  [3018] = {x=971.55, y=-22.315, z=22, rx=180, rz=141.96, shoulder=lefty, elbow=epositive, wrist=wpositive, fatherId=fReference[0]}
  [3019] = {x=972.787, y=-21.347, z=22, rx=180, rz=141.951, shoulder=lefty, elbow=epositive, wrist=wpositive, fatherId=fReference[0]}
  [3020] = {x=974.025, y=-20.378, z=22, rx=180, rz=141.942, shoulder=lefty, elbow=epositive, wrist=wpositive, fatherId=fReference[0]}
  [3021] = {x=975.263, y=-19.409, z=22, rx=180, rz=141.934, shoulder=lefty, elbow=epositive, wrist=wpositive, fatherId=fReference[0]}
  [3022] = {x=976.5, y=-18.44, z=22, rx=-180, rz=141.926, shoulder=lefty, elbow=epositive, wrist=wpositive, fatherId=fReference[0]}
  [3023] = {x=977.737, y=-17.471, z=22, rx=-180, rz=141.918, shoulder=lefty, elbow=epositive, wrist=wpositive, fatherId=fReference[0]}
  [3024] = {x=978.975, y=-16.501, z=22, rx=-180, rz=141.911, shoulder=lefty, elbow=epositive, wrist=wpositive, fatherId=fReference[0]}
  [3025] = {x=980.212, y=-15.532, z=22, rx=180, rz=141.904, shoulder=lefty, elbow=epositive, wrist=wpositive, fatherId=fReference[0]}
  [3026] = {x=981.449, y=-14.562, z=22, rx=-180, rz=141.898, shoulder=lefty, elbow=epositive, wrist=wpositive, fatherId=fReference[0]}
  [3027] = {x=982.686, y=-13.592, z=22, rx=180, rz=141.892, shoulder=lefty, elbow=epositive, wrist=wpositive, fatherId=fReference[0]}
  [3028] = {x=983.923, y=-12.621, z=22, rx=180, rz=141.887, shoulder=lefty, elbow=epositive, wrist=wpositive, fatherId=fReference[0]}
  [3029] = {x=985.16, y=-11.651, z=22, rx=-180, rz=141.882, shoulder=lefty, elbow=epositive, wrist=wpositive, fatherId=fReference[0]}
  [3030] = {x=986.397, y=-10.681, z=22, rx=180, rz=141.877, shoulder=lefty, elbow=epositive, wrist=wpositive, fatherId=fReference[0]}
  [3031] = {x=987.634, y=-9.71, z=22, rx=180, rz=141.873, shoulder=lefty, elbow=epositive, wrist=wpositive, fatherId=fReference[0]}
  [3032] = {x=988.87, y=-8.739, z=22, rx=180, rz=141.869, shoulder=lefty, elbow=epositive, wrist=wpositive, fatherId=fReference[0]}
  [3033] = {x=990.107, y=-7.769, z=22, rx=-180, rz=141.866, shoulder=lefty, elbow=epositive, wrist=wpositive, fatherId=fReference[0]}
  [3034] = {x=991.344, y=-6.798, z=22, rx=180, rz=141.863, shoulder=lefty, elbow=epositive, wrist=wpositive, fatherId=fReference[0]}
  [3035] = {x=992.58, y=-5.827, z=22, rx=-180, rz=141.86, shoulder=lefty, elbow=epositive, wrist=wpositive, fatherId=fReference[0]}
  [3036] = {x=993.817, y=-4.856, z=22, rx=180, rz=141.858, shoulder=lefty, elbow=epositive, wrist=wpositive, fatherId=fReference[0]}
  [3037] = {x=995.054, y=-3.885, z=22, rx=180, rz=141.857, shoulder=lefty, elbow=epositive, wrist=wpositive, fatherId=fReference[0]}
  [3038] = {x=996.29, y=-2.914, z=22, rx=-180, rz=141.855, shoulder=lefty, elbow=epositive, wrist=wpositive, fatherId=fReference[0]}
  [3039] = {x=997.527, y=-1.942, z=22, rx=-180, rz=141.854, shoulder=lefty, elbow=epositive, wrist=wpositive, fatherId=fReference[0]}
  [3040] = {x=998.763, y=-0.971, z=22, rx=180, rz=141.854, shoulder=lefty, elbow=epositive, wrist=wpositive, fatherId=fReference[0]}
  [3041] = {x=1000, z=22, rx=180, rz=141.854, shoulder=lefty, elbow=epositive, wrist=wpositive, fatherId=fReference[0]}
  [3042] = {x=1000, z=22, rx=180, rz=141.854, shoulder=lefty, elbow=epositive, wrist=wpositive, fatherId=fReference[0]}
  [3043] = {x=1000, z=122, rx=-180, rz=141.854, shoulder=lefty, elbow=epositive, wrist=wpositive, fatherId=fReference[0]}
  [3044] = {x=-1000, z=144, rx=180, rz=141.854, shoulder=lefty, elbow=epositive, wrist=wpositive, fatherId=fReference[0]}
  [3045] = {x=-1000, z=44, rx=180, rz=141.854, shoulder=lefty, elbow=epositive, wrist=wpositive, fatherId=fReference[0]}
  [3046] = {x=-1000, z=44, rx=180, rz=141.854, shoulder=lefty, elbow=epositive, wrist=wpositive, fatherId=fReference[0]}
  [3047] = {x=-998.763, y=0.971, z=44, rx=180, rz=141.854, shoulder=lefty, elbow=epositive, wrist=wpositive, fatherId=fReference[0]}
  [3048] = {x=-997.527, y=1.942, z=44, rx=180, rz=141.855, shoulder=lefty, elbow=epositive, wrist=wpositive, fatherId=fReference[0]}
  [3049] = {x=-996.29, y=2.914, z=44, rx=180, rz=141.857, shoulder=lefty, elbow=epositive, wrist=wpositive, fatherId=fReference[0]}
  [3050] = {x=-995.054, y=3.885, z=44, rx=180, rz=141.858, shoulder=lefty, elbow=epositive, wrist=wpositive, fatherId=fReference[0]}
  [3051] = {x=-993.817, y=4.856, z=44, rx=180, rz=141.86, shoulder=lefty, elbow=epositive, wrist=wpositive, fatherId=fReference[0]}
  [3052] = {x=-992.58, y=5.827, z=44, rx=180, rz=141.863, shoulder=lefty, elbow=epositive, wrist=wpositive, fatherId=fReference[0]}
  [3053] = {x=-991.344, y=6.798, z=44, rx=180, rz=141.866, shoulder=lefty, elbow=epositive, wrist=wpositive, fatherId=fReference[0]}
  [3054] = {x=-990.107, y=7.769, z=44, rx=180, rz=141.869, shoulder=lefty, elbow=epositive, wrist=wpositive, fatherId=fReference[0]}
  [3055] = {x=-988.87, y=8.739, z=44, rx=180, rz=141.873, shoulder=lefty, elbow=epositive, wrist=wpositive, fatherId=fReference[0]}
  [3056] = {x=-987.634, y=9.71, z=44, rx=180, rz=141.877, shoulder=lefty, elbow=epositive, wrist=wpositive, fatherId=fReference[0]}
  [3057] = {x=-986.397, y=10.681, z=44, rx=180, rz=141.882, shoulder=lefty, elbow=epositive, wrist=wpositive, fatherId=fReference[0]}
  [3058] = {x=-985.16, y=11.651, z=44, rx=180, rz=141.887, shoulder=lefty, elbow=epositive, wrist=wpositive, fatherId=fReference[0]}
  [3059] = {x=-983.923, y=12.622, z=44, rx=180, rz=141.892, shoulder=lefty, elbow=epositive, wrist=wpositive, fatherId=fReference[0]}
  [3060] = {x=-982.686, y=13.592, z=44, rx=180, rz=141.898, shoulder=lefty, elbow=epositive, wrist=wpositive, fatherId=fReference[0]}
  [3061] = {x=-981.449, y=14.562, z=44, rx=180, rz=141.904, shoulder=lefty, elbow=epositive, wrist=wpositive, fatherId=fReference[0]}
  [3062] = {x=-980.211, y=15.532, z=44, rx=180, rz=141.911, shoulder=lefty, elbow=epositive, wrist=wpositive, fatherId=fReference[0]}
  [3063] = {x=-978.974, y=16.502, z=44, rx=180, rz=141.918, shoulder=lefty, elbow=epositive, wrist=wpositive, fatherId=fReference[0]}
  [3064] = {x=-977.737, y=17.471, z=44, rx=180, rz=141.926, shoulder=lefty, elbow=epositive, wrist=wpositive, fatherId=fReference[0]}
  [3065] = {x=-976.499, y=18.441, z=44, rx=180, rz=141.934, shoulder=lefty, elbow=epositive, wrist=wpositive, fatherId=fReference[0]}
  [3066] = {x=-975.262, y=19.41, z=44, rx=180, rz=141.942, shoulder=lefty, elbow=epositive, wrist=wpositive, fatherId=fReference[0]}
  [3067] = {x=-974.024, y=20.379, z=44, rx=180, rz=141.951, shoulder=lefty, elbow=epositive, wrist=wpositive, fatherId=fReference[0]}
  [3068] = {x=-972.786, y=21.347, z=44, rx=180, rz=141.96, shoulder=lefty, elbow=epositive, wrist=wpositive, fatherId=fReference[0]}
  [3069] = {x=-971.549, y=22.316, z=44, rx=180, rz=141.97, shoulder=lefty, elbow=epositive, wrist=wpositive, fatherId=fReference[0]}
  [3070] = {x=-970.311, y=23.284, z=44, rx=180, rz=141.98, shoulder=lefty, elbow=epositive, wrist=wpositive, fatherId=fReference[0]}
  [3071] = {x=-969.072, y=24.252, z=44, rx=180, rz=141.991, shoulder=lefty, elbow=epositive, wrist=wpositive, fatherId=fReference[0]}
  [3072] = {x=-967.834, y=25.22, z=44, rx=180, rz=142.002, shoulder=lefty, elbow=epositive, wrist=wpositive, fatherId=fReference[0]}
  [3073] = {x=-966.596, y=26.187, z=44, rx=180, rz=142.013, shoulder=lefty, elbow=epositive, wrist=wpositive, fatherId=fReference[0]}
  [3074] = {x=-965.357, y=27.155, z=44, rx=180, rz=142.025, shoulder=lefty, elbow=epositive, wrist=wpositive, fatherId=fReference[0]}
  [3075] = {x=-964.119, y=28.121, z=44, rx=180, rz=142.037, shoulder=lefty, elbow=epositive, wrist=wpositive, fatherId=fReference[0]}
  [3076] = {x=-962.88, y=29.088, z=44, rx=180, rz=142.05, shoulder=lefty, elbow=epositive, wrist=wpositive, fatherId=fReference[0]}
  [3077] = {x=-961.641, y=30.054, z=44, rx=180, rz=142.063, shoulder=lefty, elbow=epositive, wrist=wpositive, fatherId=fReference[0]}
  [3078] = {x=-960.402, y=31.02, z=44, rx=180, rz=142.076, shoulder=lefty, elbow=epositive, wrist=wpositive, fatherId=fReference[0]}
  [3079] = {x=-959.163, y=31.986, z=44, rx=180, rz=142.09, shoulder=lefty, elbow=epositive, wrist=wpositive, fatherId=fReference[0]}
  [3080] = {x=-957.923, y=32.951, z=44, rx=180, rz=142.105, shoulder=lefty, elbow=epositive, wrist=wpositive, fatherId=fReference[0]}
  [3081] = {x=-956.684, y=33.916, z=44, rx=180, rz=142.12, shoulder=lefty, elbow=epositive, wrist=wpositive, fatherId=fReference[0]}
  [3082] = {x=-955.444, y=34.88, z=44, rx=180, rz=142.135, shoulder=lefty, elbow=epositive, wrist=wpositive, fatherId=fReference[0]}
  [3083] = {x=-954.204, y=35.844, z=44, rx=180, rz=142.151, shoulder=lefty, elbow=epositive, wrist=wpositive, fatherId=fReference[0]}
  [3084] = {x=-952.964, y=36.808, z=44, rx=180, rz=142.167, shoulder=lefty, elbow=epositive, wrist=wpositive, fatherId=fReference[0]}
  [3085] = {x=-951.724, y=37.771, z=44, rx=180, rz=142.183, shoulder=lefty, elbow=epositive, wrist=wpositive, fatherId=fReference[0]}
  [3086] = {x=-950.483, y=38.734, z=44, rx=180, rz=142.2, shoulder=lefty, elbow=epositive, wrist=wpositive, fatherId=fReference[0]}
  [3087] = {x=-949.243, y=39.696, z=44, rx=180, rz=142.218, shoulder=lefty, elbow=epositive, wrist=wpositive, fatherId=fReference[0]}
  [3088] = {x=-948.002, y=40.658, z=44, rx=180, rz=142.235, shoulder=lefty, elbow=epositive, wrist=wpositive, fatherId=fReference[0]}
  [3089] = {x=-946.761, y=41.619, z=44, rx=180, rz=142.254, shoulder=lefty, elbow=epositive, wrist=wpositive, fatherId=fReference[0]}
  [3090] = {x=-945.52, y=42.58, z=44, rx=180, rz=142.272, shoulder=lefty, elbow=epositive, wrist=wpositive, fatherId=fReference[0]}
  [3091] = {x=-944.278, y=43.541, z=44, rx=180, rz=142.291, shoulder=lefty, elbow=epositive, wrist=wpositive, fatherId=fReference[0]}
  [3092] = {x=-943.037, y=44.501, z=44, rx=180, rz=142.311, shoulder=lefty, elbow=epositive, wrist=wpositive, fatherId=fReference[0]}
  [3093] = {x=-941.795, y=45.46, z=44, rx=180, rz=142.331, shoulder=lefty, elbow=epositive, wrist=wpositive, fatherId=fReference[0]}
  [3094] = {x=-940.553, y=46.419, z=44, rx=180, rz=142.351, shoulder=lefty, elbow=epositive, wrist=wpositive, fatherId=fReference[0]}
  [3095] = {x=-939.31, y=47.377, z=44, rx=180, rz=142.372, shoulder=lefty, elbow=epositive, wrist=wpositive, fatherId=fReference[0]}
  [3096] = {x=-938.068, y=48.335, z=44, rx=180, rz=142.394, shoulder=lefty, elbow=epositive, wrist=wpositive, fatherId=fReference[0]}
  [3097] = {x=-936.825, y=49.292, z=44, rx=180, rz=142.415, shoulder=lefty, elbow=epositive, wrist=wpositive, fatherId=fReference[0]}
  [3098] = {x=-935.582, y=50.249, z=44, rx=180, rz=142.438, shoulder=lefty, elbow=epositive, wrist=wpositive, fatherId=fReference[0]}
  [3099] = {x=-934.339, y=51.205, z=44, rx=180, rz=142.46, shoulder=lefty, elbow=epositive, wrist=wpositive, fatherId=fReference[0]}
  [3100] = {x=-933.095, y=52.161, z=44, rx=180, rz=142.483, shoulder=lefty, elbow=epositive, wrist=wpositive, fatherId=fReference[0]}
  [3101] = {x=-931.852, y=53.116, z=44, rx=180, rz=142.507, shoulder=lefty, elbow=epositive, wrist=wpositive, fatherId=fReference[0]}
  [3102] = {x=-930.608, y=54.07, z=44, rx=-180, rz=142.531, shoulder=lefty, elbow=epositive, wrist=wpositive, fatherId=fReference[0]}
  [3103] = {x=-929.363, y=55.024, z=44, rx=180, rz=142.555, shoulder=lefty, elbow=epositive, wrist=wpositive, fatherId=fReference[0]}
  [3104] = {x=-928.119, y=55.977, z=44, rx=180, rz=142.58, shoulder=lefty, elbow=epositive, wrist=wpositive, fatherId=fReference[0]}
  [3105] = {x=-926.874, y=56.929, z=44, rx=180, rz=142.605, shoulder=lefty, elbow=epositive, wrist=wpositive, fatherId=fReference[0]}
  [3106] = {x=-925.629, y=57.881, z=44, rx=180, rz=142.631, shoulder=lefty, elbow=epositive, wrist=wpositive, fatherId=fReference[0]}
  [3107] = {x=-924.384, y=58.832, z=44, rx=180, rz=142.657, shoulder=lefty, elbow=epositive, wrist=wpositive, fatherId=fReference[0]}
  [3108] = {x=-923.138, y=59.782, z=44, rx=180, rz=142.684, shoulder=lefty, elbow=epositive, wrist=wpositive, fatherId=fReference[0]}
  [3109] = {x=-921.892, y=60.732, z=44, rx=180, rz=142.711, shoulder=lefty, elbow=epositive, wrist=wpositive, fatherId=fReference[0]}
  [3110] = {x=-920.646, y=61.681, z=44, rx=180, rz=142.738, shoulder=lefty, elbow=epositive, wrist=wpositive, fatherId=fReference[0]}
  [3111] = {x=-919.4, y=62.629, z=44, rx=180, rz=142.766, shoulder=lefty, elbow=epositive, wrist=wpositive, fatherId=fReference[0]}
  [3112] = {x=-918.153, y=63.576, z=44, rx=180, rz=142.795, shoulder=lefty, elbow=epositive, wrist=wpositive, fatherId=fReference[0]}
  [3113] = {x=-916.906, y=64.523, z=44, rx=180, rz=142.824, shoulder=lefty, elbow=epositive, wrist=wpositive, fatherId=fReference[0]}
  [3114] = {x=-915.659, y=65.469, z=44, rx=180, rz=142.853, shoulder=lefty, elbow=epositive, wrist=wpositive, fatherId=fReference[0]}
  [3115] = {x=-914.411, y=66.414, z=44, rx=180, rz=142.883, shoulder=lefty, elbow=epositive, wrist=wpositive, fatherId=fReference[0]}
  [3116] = {x=-913.163, y=67.358, z=44, rx=180, rz=142.913, shoulder=lefty, elbow=epositive, wrist=wpositive, fatherId=fReference[0]}
  [3117] = {x=-911.915, y=68.302, z=44, rx=180, rz=142.944, shoulder=lefty, elbow=epositive, wrist=wpositive, fatherId=fReference[0]}
  [3118] = {x=-910.667, y=69.245, z=44, rx=180, rz=142.975, shoulder=lefty, elbow=epositive, wrist=wpositive, fatherId=fReference[0]}
  [3119] = {x=-909.418, y=70.187, z=44, rx=180, rz=143.007, shoulder=lefty, elbow=epositive, wrist=wpositive, fatherId=fReference[0]}
  [3120] = {x=-908.169, y=71.128, z=44, rx=180, rz=143.039, shoulder=lefty, elbow=epositive, wrist=wpositive, fatherId=fReference[0]}
  [3121] = {x=-906.919, y=72.068, z=44, rx=180, rz=143.071, shoulder=lefty, elbow=epositive, wrist=wpositive, fatherId=fReference[0]}
  [3122] = {x=-905.67, y=73.007, z=44, rx=180, rz=143.104, shoulder=lefty, elbow=epositive, wrist=wpositive, fatherId=fReference[0]}
  [3123] = {x=-904.419, y=73.946, z=44, rx=180, rz=143.138, shoulder=lefty, elbow=epositive, wrist=wpositive, fatherId=fReference[0]}
  [3124] = {x=-903.169, y=74.883, z=44, rx=180, rz=143.172, shoulder=lefty, elbow=epositive, wrist=wpositive, fatherId=fReference[0]}
  [3125] = {x=-901.918, y=75.82, z=44, rx=180, rz=143.206, shoulder=lefty, elbow=epositive, wrist=wpositive, fatherId=fReference[0]}
  [3126] = {x=-900.667, y=76.756, z=44, rx=180, rz=143.241, shoulder=lefty, elbow=epositive, wrist=wpositive, fatherId=fReference[0]}
  [3127] = {x=-899.416, y=77.691, z=44, rx=180, rz=143.276, shoulder=lefty, elbow=epositive, wrist=wpositive, fatherId=fReference[0]}
  [3128] = {x=-898.164, y=78.625, z=44, rx=180, rz=143.312, shoulder=lefty, elbow=epositive, wrist=wpositive, fatherId=fReference[0]}
  [3129] = {x=-896.912, y=79.557, z=44, rx=180, rz=143.348, shoulder=lefty, elbow=epositive, wrist=wpositive, fatherId=fReference[0]}
  [3130] = {x=-895.659, y=80.489, z=44, rx=180, rz=143.385, shoulder=lefty, elbow=epositive, wrist=wpositive, fatherId=fReference[0]}
  [3131] = {x=-894.406, y=81.42, z=44, rx=180, rz=143.422, shoulder=lefty, elbow=epositive, wrist=wpositive, fatherId=fReference[0]}
  [3132] = {x=-893.153, y=82.35, z=44, rx=180, rz=143.46, shoulder=lefty, elbow=epositive, wrist=wpositive, fatherId=fReference[0]}
  [3133] = {x=-891.899, y=83.279, z=44, rx=180, rz=143.498, shoulder=lefty, elbow=epositive, wrist=wpositive, fatherId=fReference[0]}
  [3134] = {x=-890.645, y=84.207, z=44, rx=180, rz=143.536, shoulder=lefty, elbow=epositive, wrist=wpositive, fatherId=fReference[0]}
  [3135] = {x=-889.391, y=85.134, z=44, rx=180, rz=143.575, shoulder=lefty, elbow=epositive, wrist=wpositive, fatherId=fReference[0]}
  [3136] = {x=-888.136, y=86.06, z=44, rx=180, rz=143.615, shoulder=lefty, elbow=epositive, wrist=wpositive, fatherId=fReference[0]}
  [3137] = {x=-886.881, y=86.985, z=44, rx=180, rz=143.655, shoulder=lefty, elbow=epositive, wrist=wpositive, fatherId=fReference[0]}
  [3138] = {x=-885.626, y=87.909, z=44, rx=180, rz=143.696, shoulder=lefty, elbow=epositive, wrist=wpositive, fatherId=fReference[0]}
  [3139] = {x=-884.37, y=88.832, z=44, rx=180, rz=143.737, shoulder=lefty, elbow=epositive, wrist=wpositive, fatherId=fReference[0]}
  [3140] = {x=-883.113, y=89.753, z=44, rx=180, rz=143.778, shoulder=lefty, elbow=epositive, wrist=wpositive, fatherId=fReference[0]}
  [3141] = {x=-881.857, y=90.674, z=44, rx=180, rz=143.82, shoulder=lefty, elbow=epositive, wrist=wpositive, fatherId=fReference[0]}
  [3142] = {x=-880.6, y=91.593, z=44, rx=180, rz=143.862, shoulder=lefty, elbow=epositive, wrist=wpositive, fatherId=fReference[0]}
  [3143] = {x=-879.342, y=92.511, z=44, rx=180, rz=143.905, shoulder=lefty, elbow=epositive, wrist=wpositive, fatherId=fReference[0]}
  [3144] = {x=-878.084, y=93.428, z=44, rx=180, rz=143.949, shoulder=lefty, elbow=epositive, wrist=wpositive, fatherId=fReference[0]}
  [3145] = {x=-876.826, y=94.344, z=44, rx=180, rz=143.993, shoulder=lefty, elbow=epositive, wrist=wpositive, fatherId=fReference[0]}
  [3146] = {x=-875.567, y=95.259, z=44, rx=180, rz=144.037, shoulder=lefty, elbow=epositive, wrist=wpositive, fatherId=fReference[0]}
  [3147] = {x=-874.308, y=96.173, z=44, rx=180, rz=144.082, shoulder=lefty, elbow=epositive, wrist=wpositive, fatherId=fReference[0]}
  [3148] = {x=-873.049, y=97.085, z=44, rx=180, rz=144.127, shoulder=lefty, elbow=epositive, wrist=wpositive, fatherId=fReference[0]}
  [3149] = {x=-871.789, y=97.996, z=44, rx=180, rz=144.173, shoulder=lefty, elbow=epositive, wrist=wpositive, fatherId=fReference[0]}
  [3150] = {x=-870.528, y=98.906, z=44, rx=180, rz=144.22, shoulder=lefty, elbow=epositive, wrist=wpositive, fatherId=fReference[0]}
  [3151] = {x=-869.267, y=99.815, z=44, rx=-180, rz=144.266, shoulder=lefty, elbow=epositive, wrist=wpositive, fatherId=fReference[0]}
  [3152] = {x=-868.006, y=100.722, z=44, rx=180, rz=144.314, shoulder=lefty, elbow=epositive, wrist=wpositive, fatherId=fReference[0]}
  [3153] = {x=-866.745, y=101.628, z=44, rx=180, rz=144.362, shoulder=lefty, elbow=epositive, wrist=wpositive, fatherId=fReference[0]}
  [3154] = {x=-865.482, y=102.533, z=44, rx=180, rz=144.41, shoulder=lefty, elbow=epositive, wrist=wpositive, fatherId=fReference[0]}
  [3155] = {x=-864.22, y=103.437, z=44, rx=180, rz=144.459, shoulder=lefty, elbow=epositive, wrist=wpositive, fatherId=fReference[0]}
  [3156] = {x=-862.957, y=104.339, z=44, rx=180, rz=144.508, shoulder=lefty, elbow=epositive, wrist=wpositive, fatherId=fReference[0]}
  [3157] = {x=-861.693, y=105.24, z=44, rx=180, rz=144.558, shoulder=lefty, elbow=epositive, wrist=wpositive, fatherId=fReference[0]}
  [3158] = {x=-860.429, y=106.139, z=44, rx=180, rz=144.609, shoulder=lefty, elbow=epositive, wrist=wpositive, fatherId=fReference[0]}
  [3159] = {x=-859.165, y=107.038, z=44, rx=180, rz=144.659, shoulder=lefty, elbow=epositive, wrist=wpositive, fatherId=fReference[0]}
  [3160] = {x=-857.9, y=107.935, z=44, rx=180, rz=144.711, shoulder=lefty, elbow=epositive, wrist=wpositive, fatherId=fReference[0]}
  [3161] = {x=-856.635, y=108.83, z=44, rx=180, rz=144.763, shoulder=lefty, elbow=epositive, wrist=wpositive, fatherId=fReference[0]}
  [3162] = {x=-855.369, y=109.724, z=44, rx=180, rz=144.815, shoulder=lefty, elbow=epositive, wrist=wpositive, fatherId=fReference[0]}
  [3163] = {x=-854.103, y=110.617, z=44, rx=180, rz=144.868, shoulder=lefty, elbow=epositive, wrist=wpositive, fatherId=fReference[0]}
  [3164] = {x=-852.836, y=111.508, z=44, rx=180, rz=144.922, shoulder=lefty, elbow=epositive, wrist=wpositive, fatherId=fReference[0]}
  [3165] = {x=-851.569, y=112.398, z=44, rx=180, rz=144.976, shoulder=lefty, elbow=epositive, wrist=wpositive, fatherId=fReference[0]}
  [3166] = {x=-850.301, y=113.287, z=44, rx=180, rz=145.03, shoulder=lefty, elbow=epositive, wrist=wpositive, fatherId=fReference[0]}
  [3167] = {x=-849.033, y=114.174, z=44, rx=180, rz=145.085, shoulder=lefty, elbow=epositive, wrist=wpositive, fatherId=fReference[0]}
  [3168] = {x=-847.764, y=115.059, z=44, rx=180, rz=145.141, shoulder=lefty, elbow=epositive, wrist=wpositive, fatherId=fReference[0]}
  [3169] = {x=-846.495, y=115.943, z=44, rx=180, rz=145.197, shoulder=lefty, elbow=epositive, wrist=wpositive, fatherId=fReference[0]}
  [3170] = {x=-845.225, y=116.826, z=44, rx=180, rz=145.253, shoulder=lefty, elbow=epositive, wrist=wpositive, fatherId=fReference[0]}
  [3171] = {x=-843.955, y=117.707, z=44, rx=180, rz=145.311, shoulder=lefty, elbow=epositive, wrist=wpositive, fatherId=fReference[0]}
  [3172] = {x=-842.685, y=118.586, z=44, rx=180, rz=145.368, shoulder=lefty, elbow=epositive, wrist=wpositive, fatherId=fReference[0]}
  [3173] = {x=-841.413, y=119.464, z=44, rx=180, rz=145.426, shoulder=lefty, elbow=epositive, wrist=wpositive, fatherId=fReference[0]}
  [3174] = {x=-840.142, y=120.341, z=44, rx=180, rz=145.485, shoulder=lefty, elbow=epositive, wrist=wpositive, fatherId=fReference[0]}
  [3175] = {x=-838.869, y=121.216, z=44, rx=180, rz=145.544, shoulder=lefty, elbow=epositive, wrist=wpositive, fatherId=fReference[0]}
  [3176] = {x=-837.597, y=122.089, z=44, rx=180, rz=145.604, shoulder=lefty, elbow=epositive, wrist=wpositive, fatherId=fReference[0]}
  [3177] = {x=-836.323, y=122.961, z=44, rx=180, rz=145.665, shoulder=lefty, elbow=epositive, wrist=wpositive, fatherId=fReference[0]}
  [3178] = {x=-835.049, y=123.831, z=44, rx=180, rz=145.725, shoulder=lefty, elbow=epositive, wrist=wpositive, fatherId=fReference[0]}
  [3179] = {x=-833.775, y=124.699, z=44, rx=180, rz=145.787, shoulder=lefty, elbow=epositive, wrist=wpositive, fatherId=fReference[0]}
  [3180] = {x=-832.5, y=125.566, z=44, rx=180, rz=145.849, shoulder=lefty, elbow=epositive, wrist=wpositive, fatherId=fReference[0]}
  [3181] = {x=-831.225, y=126.431, z=44, rx=180, rz=145.911, shoulder=lefty, elbow=epositive, wrist=wpositive, fatherId=fReference[0]}
  [3182] = {x=-829.949, y=127.295, z=44, rx=180, rz=145.974, shoulder=lefty, elbow=epositive, wrist=wpositive, fatherId=fReference[0]}
  [3183] = {x=-828.672, y=128.157, z=44, rx=180, rz=146.038, shoulder=lefty, elbow=epositive, wrist=wpositive, fatherId=fReference[0]}
  [3184] = {x=-827.395, y=129.017, z=44, rx=180, rz=146.102, shoulder=lefty, elbow=epositive, wrist=wpositive, fatherId=fReference[0]}
  [3185] = {x=-826.117, y=129.876, z=44, rx=180, rz=146.167, shoulder=lefty, elbow=epositive, wrist=wpositive, fatherId=fReference[0]}
  [3186] = {x=-824.839, y=130.732, z=44, rx=180, rz=146.232, shoulder=lefty, elbow=epositive, wrist=wpositive, fatherId=fReference[0]}
  [3187] = {x=-823.56, y=131.587, z=44, rx=180, rz=146.298, shoulder=lefty, elbow=epositive, wrist=wpositive, fatherId=fReference[0]}
  [3188] = {x=-822.281, y=132.441, z=44, rx=180, rz=146.364, shoulder=lefty, elbow=epositive, wrist=wpositive, fatherId=fReference[0]}
  [3189] = {x=-821.001, y=133.292, z=44, rx=180, rz=146.431, shoulder=lefty, elbow=epositive, wrist=wpositive, fatherId=fReference[0]}
  [3190] = {x=-819.721, y=134.142, z=44, rx=180, rz=146.499, shoulder=lefty, elbow=epositive, wrist=wpositive, fatherId=fReference[0]}
  [3191] = {x=-818.44, y=134.99, z=44, rx=180, rz=146.567, shoulder=lefty, elbow=epositive, wrist=wpositive, fatherId=fReference[0]}
  [3192] = {x=-817.158, y=135.836, z=44, rx=180, rz=146.636, shoulder=lefty, elbow=epositive, wrist=wpositive, fatherId=fReference[0]}
  [3193] = {x=-815.876, y=136.68, z=44, rx=180, rz=146.705, shoulder=lefty, elbow=epositive, wrist=wpositive, fatherId=fReference[0]}
  [3194] = {x=-814.593, y=137.523, z=44, rx=180, rz=146.775, shoulder=lefty, elbow=epositive, wrist=wpositive, fatherId=fReference[0]}
  [3195] = {x=-813.309, y=138.364, z=44, rx=180, rz=146.845, shoulder=lefty, elbow=epositive, wrist=wpositive, fatherId=fReference[0]}
  [3196] = {x=-812.025, y=139.202, z=44, rx=180, rz=146.916, shoulder=lefty, elbow=epositive, wrist=wpositive, fatherId=fReference[0]}
  [3197] = {x=-810.74, y=140.039, z=44, rx=180, rz=146.987, shoulder=lefty, elbow=epositive, wrist=wpositive, fatherId=fReference[0]}
  [3198] = {x=-809.455, y=140.875, z=44, rx=180, rz=147.059, shoulder=lefty, elbow=epositive, wrist=wpositive, fatherId=fReference[0]}
  [3199] = {x=-808.169, y=141.708, z=44, rx=180, rz=147.132, shoulder=lefty, elbow=epositive, wrist=wpositive, fatherId=fReference[0]}
  [3200] = {x=-806.883, y=142.539, z=44, rx=180, rz=147.205, shoulder=lefty, elbow=epositive, wrist=wpositive, fatherId=fReference[0]}
  [3201] = {x=-805.596, y=143.368, z=44, rx=180, rz=147.279, shoulder=lefty, elbow=epositive, wrist=wpositive, fatherId=fReference[0]}
  [3202] = {x=-804.308, y=144.196, z=44, rx=180, rz=147.353, shoulder=lefty, elbow=epositive, wrist=wpositive, fatherId=fReference[0]}
  [3203] = {x=-803.019, y=145.021, z=44, rx=180, rz=147.428, shoulder=lefty, elbow=epositive, wrist=wpositive, fatherId=fReference[0]}
  [3204] = {x=-801.73, y=145.845, z=44, rx=180, rz=147.504, shoulder=lefty, elbow=epositive, wrist=wpositive, fatherId=fReference[0]}
  [3205] = {x=-800.44, y=146.666, z=44, rx=180, rz=147.58, shoulder=lefty, elbow=epositive, wrist=wpositive, fatherId=fReference[0]}
  [3206] = {x=-799.15, y=147.486, z=44, rx=180, rz=147.657, shoulder=lefty, elbow=epositive, wrist=wpositive, fatherId=fReference[0]}
  [3207] = {x=-797.859, y=148.303, z=44, rx=180, rz=147.734, shoulder=lefty, elbow=epositive, wrist=wpositive, fatherId=fReference[0]}
  [3208] = {x=-796.567, y=149.119, z=44, rx=180, rz=147.812, shoulder=lefty, elbow=epositive, wrist=wpositive, fatherId=fReference[0]}
  [3209] = {x=-795.275, y=149.932, z=44, rx=180, rz=147.891, shoulder=lefty, elbow=epositive, wrist=wpositive, fatherId=fReference[0]}
  [3210] = {x=-793.982, y=150.744, z=44, rx=180, rz=147.97, shoulder=lefty, elbow=epositive, wrist=wpositive, fatherId=fReference[0]}
  [3211] = {x=-792.688, y=151.553, z=44, rx=180, rz=148.05, shoulder=lefty, elbow=epositive, wrist=wpositive, fatherId=fReference[0]}
  [3212] = {x=-791.394, y=152.36, z=44, rx=180, rz=148.13, shoulder=lefty, elbow=epositive, wrist=wpositive, fatherId=fReference[0]}
  [3213] = {x=-790.099, y=153.165, z=44, rx=180, rz=148.211, shoulder=lefty, elbow=epositive, wrist=wpositive, fatherId=fReference[0]}
  [3214] = {x=-788.803, y=153.968, z=44, rx=180, rz=148.293, shoulder=lefty, elbow=epositive, wrist=wpositive, fatherId=fReference[0]}
  [3215] = {x=-787.507, y=154.769, z=44, rx=180, rz=148.375, shoulder=lefty, elbow=epositive, wrist=wpositive, fatherId=fReference[0]}
  [3216] = {x=-786.21, y=155.568, z=44, rx=180, rz=148.458, shoulder=lefty, elbow=epositive, wrist=wpositive, fatherId=fReference[0]}
  [3217] = {x=-784.912, y=156.365, z=44, rx=180, rz=148.541, shoulder=lefty, elbow=epositive, wrist=wpositive, fatherId=fReference[0]}
  [3218] = {x=-783.613, y=157.159, z=44, rx=180, rz=148.625, shoulder=lefty, elbow=epositive, wrist=wpositive, fatherId=fReference[0]}
  [3219] = {x=-782.314, y=157.951, z=44, rx=180, rz=148.71, shoulder=lefty, elbow=epositive, wrist=wpositive, fatherId=fReference[0]}
  [3220] = {x=-781.014, y=158.741, z=44, rx=180, rz=148.795, shoulder=lefty, elbow=epositive, wrist=wpositive, fatherId=fReference[0]}
  [3221] = {x=-779.714, y=159.529, z=44, rx=180, rz=148.881, shoulder=lefty, elbow=epositive, wrist=wpositive, fatherId=fReference[0]}
  [3222] = {x=-778.413, y=160.315, z=44, rx=180, rz=148.968, shoulder=lefty, elbow=epositive, wrist=wpositive, fatherId=fReference[0]}
  [3223] = {x=-777.111, y=161.098, z=44, rx=180, rz=149.055, shoulder=lefty, elbow=epositive, wrist=wpositive, fatherId=fReference[0]}
  [3224] = {x=-775.808, y=161.879, z=44, rx=180, rz=149.143, shoulder=lefty, elbow=epositive, wrist=wpositive, fatherId=fReference[0]}
  [3225] = {x=-774.505, y=162.658, z=44, rx=180, rz=149.231, shoulder=lefty, elbow=epositive, wrist=wpositive, fatherId=fReference[0]}
  [3226] = {x=-773.2, y=163.434, z=44, rx=180, rz=149.32, shoulder=lefty, elbow=epositive, wrist=wpositive, fatherId=fReference[0]}
  [3227] = {x=-771.896, y=164.208, z=44, rx=180, rz=149.41, shoulder=lefty, elbow=epositive, wrist=wpositive, fatherId=fReference[0]}
  [3228] = {x=-770.59, y=164.98, z=44, rx=180, rz=149.5, shoulder=lefty, elbow=epositive, wrist=wpositive, fatherId=fReference[0]}
  [3229] = {x=-769.284, y=165.75, z=44, rx=-180, rz=149.591, shoulder=lefty, elbow=epositive, wrist=wpositive, fatherId=fReference[0]}
  [3230] = {x=-767.977, y=166.517, z=44, rx=180, rz=149.683, shoulder=lefty, elbow=epositive, wrist=wpositive, fatherId=fReference[0]}
  [3231] = {x=-766.669, y=167.281, z=44, rx=180, rz=149.775, shoulder=lefty, elbow=epositive, wrist=wpositive, fatherId=fReference[0]}
  [3232] = {x=-765.36, y=168.044, z=44, rx=180, rz=149.868, shoulder=lefty, elbow=epositive, wrist=wpositive, fatherId=fReference[0]}
  [3233] = {x=-764.051, y=168.804, z=44, rx=180, rz=149.962, shoulder=lefty, elbow=epositive, wrist=wpositive, fatherId=fReference[0]}
  [3234] = {x=-762.741, y=169.561, z=44, rx=180, rz=150.056, shoulder=lefty, elbow=epositive, wrist=wpositive, fatherId=fReference[0]}
  [3235] = {x=-761.431, y=170.316, z=44, rx=180, rz=150.151, shoulder=lefty, elbow=epositive, wrist=wpositive, fatherId=fReference[0]}
  [3236] = {x=-760.119, y=171.069, z=44, rx=180, rz=150.247, shoulder=lefty, elbow=epositive, wrist=wpositive, fatherId=fReference[0]}
  [3237] = {x=-758.807, y=171.819, z=44, rx=-180, rz=150.343, shoulder=lefty, elbow=epositive, wrist=wpositive, fatherId=fReference[0]}
  [3238] = {x=-757.494, y=172.566, z=44, rx=180, rz=150.44, shoulder=lefty, elbow=epositive, wrist=wpositive, fatherId=fReference[0]}
  [3239] = {x=-756.181, y=173.311, z=44, rx=180, rz=150.537, shoulder=lefty, elbow=epositive, wrist=wpositive, fatherId=fReference[0]}
  [3240] = {x=-754.866, y=174.054, z=44, rx=180, rz=150.636, shoulder=lefty, elbow=epositive, wrist=wpositive, fatherId=fReference[0]}
  [3241] = {x=-753.551, y=174.794, z=44, rx=180, rz=150.734, shoulder=lefty, elbow=epositive, wrist=wpositive, fatherId=fReference[0]}
  [3242] = {x=-752.235, y=175.531, z=44, rx=-180, rz=150.834, shoulder=lefty, elbow=epositive, wrist=wpositive, fatherId=fReference[0]}
  [3243] = {x=-750.919, y=176.266, z=44, rx=-180, rz=150.934, shoulder=lefty, elbow=epositive, wrist=wpositive, fatherId=fReference[0]}
  [3244] = {x=-749.601, y=176.998, z=44, rx=180, rz=151.035, shoulder=lefty, elbow=epositive, wrist=wpositive, fatherId=fReference[0]}
  [3245] = {x=-748.283, y=177.727, z=44, rx=180, rz=151.137, shoulder=lefty, elbow=epositive, wrist=wpositive, fatherId=fReference[0]}
  [3246] = {x=-746.965, y=178.454, z=44, rx=180, rz=151.239, shoulder=lefty, elbow=epositive, wrist=wpositive, fatherId=fReference[0]}
  [3247] = {x=-745.645, y=179.179, z=44, rx=180, rz=151.342, shoulder=lefty, elbow=epositive, wrist=wpositive, fatherId=fReference[0]}
  [3248] = {x=-744.325, y=179.9, z=44, rx=-180, rz=151.445, shoulder=lefty, elbow=epositive, wrist=wpositive, fatherId=fReference[0]}
  [3249] = {x=-743.004, y=180.619, z=44, rx=180, rz=151.549, shoulder=lefty, elbow=epositive, wrist=wpositive, fatherId=fReference[0]}
  [3250] = {x=-741.682, y=181.335, z=44, rx=180, rz=151.654, shoulder=lefty, elbow=epositive, wrist=wpositive, fatherId=fReference[0]}
  [3251] = {x=-740.359, y=182.049, z=44, rx=180, rz=151.76, shoulder=lefty, elbow=epositive, wrist=wpositive, fatherId=fReference[0]}
  [3252] = {x=-739.036, y=182.76, z=44, rx=180, rz=151.866, shoulder=lefty, elbow=epositive, wrist=wpositive, fatherId=fReference[0]}
  [3253] = {x=-737.712, y=183.468, z=44, rx=180, rz=151.973, shoulder=lefty, elbow=epositive, wrist=wpositive, fatherId=fReference[0]}
  [3254] = {x=-736.387, y=184.173, z=44, rx=180, rz=152.081, shoulder=lefty, elbow=epositive, wrist=wpositive, fatherId=fReference[0]}
  [3255] = {x=-735.061, y=184.875, z=44, rx=180, rz=152.189, shoulder=lefty, elbow=epositive, wrist=wpositive, fatherId=fReference[0]}
  [3256] = {x=-733.735, y=185.575, z=44, rx=180, rz=152.298, shoulder=lefty, elbow=epositive, wrist=wpositive, fatherId=fReference[0]}
  [3257] = {x=-732.408, y=186.272, z=44, rx=180, rz=152.408, shoulder=lefty, elbow=epositive, wrist=wpositive, fatherId=fReference[0]}
  [3258] = {x=-731.08, y=186.966, z=44, rx=-180, rz=152.518, shoulder=lefty, elbow=epositive, wrist=wpositive, fatherId=fReference[0]}
  [3259] = {x=-729.751, y=187.657, z=44, rx=180, rz=152.63, shoulder=lefty, elbow=epositive, wrist=wpositive, fatherId=fReference[0]}
  [3260] = {x=-728.422, y=188.345, z=44, rx=180, rz=152.741, shoulder=lefty, elbow=epositive, wrist=wpositive, fatherId=fReference[0]}
  [3261] = {x=-727.092, y=189.03, z=44, rx=180, rz=152.854, shoulder=lefty, elbow=epositive, wrist=wpositive, fatherId=fReference[0]}
  [3262] = {x=-725.761, y=189.713, z=44, rx=180, rz=152.967, shoulder=lefty, elbow=epositive, wrist=wpositive, fatherId=fReference[0]}
  [3263] = {x=-724.429, y=190.392, z=44, rx=180, rz=153.081, shoulder=lefty, elbow=epositive, wrist=wpositive, fatherId=fReference[0]}
  [3264] = {x=-723.097, y=191.069, z=44, rx=180, rz=153.196, shoulder=lefty, elbow=epositive, wrist=wpositive, fatherId=fReference[0]}
  [3265] = {x=-721.764, y=191.742, z=44, rx=180, rz=153.311, shoulder=lefty, elbow=epositive, wrist=wpositive, fatherId=fReference[0]}
  [3266] = {x=-720.43, y=192.413, z=44, rx=180, rz=153.427, shoulder=lefty, elbow=epositive, wrist=wpositive, fatherId=fReference[0]}
  [3267] = {x=-719.095, y=193.08, z=44, rx=180, rz=153.544, shoulder=lefty, elbow=epositive, wrist=wpositive, fatherId=fReference[0]}
  [3268] = {x=-717.76, y=193.745, z=44, rx=180, rz=153.661, shoulder=lefty, elbow=epositive, wrist=wpositive, fatherId=fReference[0]}
  [3269] = {x=-716.424, y=194.406, z=44, rx=180, rz=153.779, shoulder=lefty, elbow=epositive, wrist=wpositive, fatherId=fReference[0]}
  [3270] = {x=-715.087, y=195.065, z=44, rx=180, rz=153.898, shoulder=lefty, elbow=epositive, wrist=wpositive, fatherId=fReference[0]}
  [3271] = {x=-713.749, y=195.72, z=44, rx=180, rz=154.017, shoulder=lefty, elbow=epositive, wrist=wpositive, fatherId=fReference[0]}
  [3272] = {x=-712.411, y=196.372, z=44, rx=180, rz=154.138, shoulder=lefty, elbow=epositive, wrist=wpositive, fatherId=fReference[0]}
  [3273] = {x=-711.072, y=197.022, z=44, rx=180, rz=154.259, shoulder=lefty, elbow=epositive, wrist=wpositive, fatherId=fReference[0]}
  [3274] = {x=-709.732, y=197.668, z=44, rx=180, rz=154.38, shoulder=lefty, elbow=epositive, wrist=wpositive, fatherId=fReference[0]}
  [3275] = {x=-708.391, y=198.311, z=44, rx=180, rz=154.503, shoulder=lefty, elbow=epositive, wrist=wpositive, fatherId=fReference[0]}
  [3276] = {x=-707.05, y=198.95, z=44, rx=-180, rz=154.626, shoulder=lefty, elbow=epositive, wrist=wpositive, fatherId=fReference[0]}
  [3277] = {x=-705.708, y=199.587, z=44, rx=180, rz=154.75, shoulder=lefty, elbow=epositive, wrist=wpositive, fatherId=fReference[0]}
  [3278] = {x=-704.365, y=200.22, z=44, rx=180, rz=154.874, shoulder=lefty, elbow=epositive, wrist=wpositive, fatherId=fReference[0]}
  [3279] = {x=-703.021, y=200.85, z=44, rx=180, rz=154.999, shoulder=lefty, elbow=epositive, wrist=wpositive, fatherId=fReference[0]}
  [3280] = {x=-701.677, y=201.477, z=44, rx=180, rz=155.125, shoulder=lefty, elbow=epositive, wrist=wpositive, fatherId=fReference[0]}
  [3281] = {x=-700.332, y=202.101, z=44, rx=180, rz=155.252, shoulder=lefty, elbow=epositive, wrist=wpositive, fatherId=fReference[0]}
  [3282] = {x=-698.986, y=202.721, z=44, rx=180, rz=155.379, shoulder=lefty, elbow=epositive, wrist=wpositive, fatherId=fReference[0]}
  [3283] = {x=-697.639, y=203.338, z=44, rx=180, rz=155.508, shoulder=lefty, elbow=epositive, wrist=wpositive, fatherId=fReference[0]}
  [3284] = {x=-696.292, y=203.952, z=44, rx=-180, rz=155.636, shoulder=lefty, elbow=epositive, wrist=wpositive, fatherId=fReference[0]}
  [3285] = {x=-694.944, y=204.563, z=44, rx=180, rz=155.766, shoulder=lefty, elbow=epositive, wrist=wpositive, fatherId=fReference[0]}
  [3286] = {x=-693.595, y=205.17, z=44, rx=180, rz=155.896, shoulder=lefty, elbow=epositive, wrist=wpositive, fatherId=fReference[0]}
  [3287] = {x=-692.246, y=205.774, z=44, rx=180, rz=156.027, shoulder=lefty, elbow=epositive, wrist=wpositive, fatherId=fReference[0]}
  [3288] = {x=-690.895, y=206.374, z=44, rx=180, rz=156.159, shoulder=lefty, elbow=epositive, wrist=wpositive, fatherId=fReference[0]}
  [3289] = {x=-689.544, y=206.971, z=44, rx=180, rz=156.291, shoulder=lefty, elbow=epositive, wrist=wpositive, fatherId=fReference[0]}
  [3290] = {x=-688.193, y=207.565, z=44, rx=-180, rz=156.425, shoulder=lefty, elbow=epositive, wrist=wpositive, fatherId=fReference[0]}
  [3291] = {x=-686.84, y=208.155, z=44, rx=180, rz=156.559, shoulder=lefty, elbow=epositive, wrist=wpositive, fatherId=fReference[0]}
  [3292] = {x=-685.487, y=208.741, z=44, rx=180, rz=156.693, shoulder=lefty, elbow=epositive, wrist=wpositive, fatherId=fReference[0]}
  [3293] = {x=-684.133, y=209.325, z=44, rx=180, rz=156.828, shoulder=lefty, elbow=epositive, wrist=wpositive, fatherId=fReference[0]}
  [3294] = {x=-682.778, y=209.905, z=44, rx=180, rz=156.965, shoulder=lefty, elbow=epositive, wrist=wpositive, fatherId=fReference[0]}
  [3295] = {x=-681.423, y=210.481, z=44, rx=180, rz=157.101, shoulder=lefty, elbow=epositive, wrist=wpositive, fatherId=fReference[0]}
  [3296] = {x=-680.067, y=211.054, z=44, rx=-180, rz=157.239, shoulder=lefty, elbow=epositive, wrist=wpositive, fatherId=fReference[0]}
  [3297] = {x=-678.71, y=211.623, z=44, rx=180, rz=157.377, shoulder=lefty, elbow=epositive, wrist=wpositive, fatherId=fReference[0]}
  [3298] = {x=-677.353, y=212.189, z=44, rx=-180, rz=157.516, shoulder=lefty, elbow=epositive, wrist=wpositive, fatherId=fReference[0]}
  [3299] = {x=-675.994, y=212.751, z=44, rx=-180, rz=157.656, shoulder=lefty, elbow=epositive, wrist=wpositive, fatherId=fReference[0]}
  [3300] = {x=-674.635, y=213.309, z=44, rx=180, rz=157.796, shoulder=lefty, elbow=epositive, wrist=wpositive, fatherId=fReference[0]}
  [3301] = {x=-673.276, y=213.864, z=44, rx=180, rz=157.937, shoulder=lefty, elbow=epositive, wrist=wpositive, fatherId=fReference[0]}
  [3302] = {x=-671.915, y=214.416, z=44, rx=180, rz=158.079, shoulder=lefty, elbow=epositive, wrist=wpositive, fatherId=fReference[0]}
  [3303] = {x=-670.554, y=214.963, z=44, rx=180, rz=158.222, shoulder=lefty, elbow=epositive, wrist=wpositive, fatherId=fReference[0]}
  [3304] = {x=-669.193, y=215.508, z=44, rx=180, rz=158.365, shoulder=lefty, elbow=epositive, wrist=wpositive, fatherId=fReference[0]}
  [3305] = {x=-667.83, y=216.048, z=44, rx=-180, rz=158.509, shoulder=lefty, elbow=epositive, wrist=wpositive, fatherId=fReference[0]}
  [3306] = {x=-666.467, y=216.585, z=44, rx=180, rz=158.654, shoulder=lefty, elbow=epositive, wrist=wpositive, fatherId=fReference[0]}
  [3307] = {x=-665.103, y=217.118, z=44, rx=180, rz=158.799, shoulder=lefty, elbow=epositive, wrist=wpositive, fatherId=fReference[0]}
  [3308] = {x=-663.739, y=217.647, z=44, rx=180, rz=158.945, shoulder=lefty, elbow=epositive, wrist=wpositive, fatherId=fReference[0]}
  [3309] = {x=-662.373, y=218.173, z=44, rx=180, rz=159.092, shoulder=lefty, elbow=epositive, wrist=wpositive, fatherId=fReference[0]}
  [3310] = {x=-661.007, y=218.694, z=44, rx=180, rz=159.24, shoulder=lefty, elbow=epositive, wrist=wpositive, fatherId=fReference[0]}
  [3311] = {x=-659.641, y=219.212, z=44, rx=180, rz=159.388, shoulder=lefty, elbow=epositive, wrist=wpositive, fatherId=fReference[0]}
  [3312] = {x=-658.273, y=219.727, z=44, rx=180, rz=159.537, shoulder=lefty, elbow=epositive, wrist=wpositive, fatherId=fReference[0]}
  [3313] = {x=-656.905, y=220.237, z=44, rx=180, rz=159.687, shoulder=lefty, elbow=epositive, wrist=wpositive, fatherId=fReference[0]}
  [3314] = {x=-655.537, y=220.744, z=44, rx=180, rz=159.837, shoulder=lefty, elbow=epositive, wrist=wpositive, fatherId=fReference[0]}
  [3315] = {x=-654.167, y=221.247, z=44, rx=180, rz=159.988, shoulder=lefty, elbow=epositive, wrist=wpositive, fatherId=fReference[0]}
  [3316] = {x=-652.797, y=221.746, z=44, rx=180, rz=160.14, shoulder=lefty, elbow=epositive, wrist=wpositive, fatherId=fReference[0]}
  [3317] = {x=-651.426, y=222.241, z=44, rx=180, rz=160.293, shoulder=lefty, elbow=epositive, wrist=wpositive, fatherId=fReference[0]}
  [3318] = {x=-650.055, y=222.732, z=44, rx=180, rz=160.446, shoulder=lefty, elbow=epositive, wrist=wpositive, fatherId=fReference[0]}
  [3319] = {x=-648.683, y=223.219, z=44, rx=180, rz=160.6, shoulder=lefty, elbow=epositive, wrist=wpositive, fatherId=fReference[0]}
  [3320] = {x=-647.31, y=223.703, z=44, rx=180, rz=160.755, shoulder=lefty, elbow=epositive, wrist=wpositive, fatherId=fReference[0]}
  [3321] = {x=-645.937, y=224.182, z=44, rx=180, rz=160.91, shoulder=lefty, elbow=epositive, wrist=wpositive, fatherId=fReference[0]}
  [3322] = {x=-644.562, y=224.658, z=44, rx=180, rz=161.066, shoulder=lefty, elbow=epositive, wrist=wpositive, fatherId=fReference[0]}
  [3323] = {x=-643.188, y=225.129, z=44, rx=180, rz=161.223, shoulder=lefty, elbow=epositive, wrist=wpositive, fatherId=fReference[0]}
  [3324] = {x=-641.812, y=225.597, z=44, rx=180, rz=161.381, shoulder=lefty, elbow=epositive, wrist=wpositive, fatherId=fReference[0]}
  [3325] = {x=-640.436, y=226.061, z=44, rx=-180, rz=161.539, shoulder=lefty, elbow=epositive, wrist=wpositive, fatherId=fReference[0]}
  [3326] = {x=-639.06, y=226.52, z=44, rx=180, rz=161.698, shoulder=lefty, elbow=epositive, wrist=wpositive, fatherId=fReference[0]}
  [3327] = {x=-637.682, y=226.976, z=44, rx=180, rz=161.857, shoulder=lefty, elbow=epositive, wrist=wpositive, fatherId=fReference[0]}
  [3328] = {x=-636.304, y=227.427, z=44, rx=-180, rz=162.017, shoulder=lefty, elbow=epositive, wrist=wpositive, fatherId=fReference[0]}
  [3329] = {x=-634.925, y=227.875, z=44, rx=180, rz=162.178, shoulder=lefty, elbow=epositive, wrist=wpositive, fatherId=fReference[0]}
  [3330] = {x=-633.546, y=228.318, z=44, rx=-180, rz=162.34, shoulder=lefty, elbow=epositive, wrist=wpositive, fatherId=fReference[0]}
  [3331] = {x=-632.166, y=228.758, z=44, rx=180, rz=162.502, shoulder=lefty, elbow=epositive, wrist=wpositive, fatherId=fReference[0]}
  [3332] = {x=-630.786, y=229.193, z=44, rx=180, rz=162.665, shoulder=lefty, elbow=epositive, wrist=wpositive, fatherId=fReference[0]}
  [3333] = {x=-629.404, y=229.624, z=44, rx=180, rz=162.829, shoulder=lefty, elbow=epositive, wrist=wpositive, fatherId=fReference[0]}
  [3334] = {x=-628.022, y=230.051, z=44, rx=180, rz=162.993, shoulder=lefty, elbow=epositive, wrist=wpositive, fatherId=fReference[0]}
  [3335] = {x=-626.64, y=230.474, z=44, rx=180, rz=163.158, shoulder=lefty, elbow=epositive, wrist=wpositive, fatherId=fReference[0]}
  [3336] = {x=-625.257, y=230.893, z=44, rx=-180, rz=163.324, shoulder=lefty, elbow=epositive, wrist=wpositive, fatherId=fReference[0]}
  [3337] = {x=-623.873, y=231.307, z=44, rx=180, rz=163.49, shoulder=lefty, elbow=epositive, wrist=wpositive, fatherId=fReference[0]}
  [3338] = {x=-622.489, y=231.717, z=44, rx=180, rz=163.657, shoulder=lefty, elbow=epositive, wrist=wpositive, fatherId=fReference[0]}
  [3339] = {x=-621.104, y=232.124, z=44, rx=-180, rz=163.824, shoulder=lefty, elbow=epositive, wrist=wpositive, fatherId=fReference[0]}
  [3340] = {x=-619.718, y=232.526, z=44, rx=-180, rz=163.993, shoulder=lefty, elbow=epositive, wrist=wpositive, fatherId=fReference[0]}
  [3341] = {x=-618.332, y=232.923, z=44, rx=180, rz=164.161, shoulder=lefty, elbow=epositive, wrist=wpositive, fatherId=fReference[0]}
  [3342] = {x=-616.945, y=233.317, z=44, rx=180, rz=164.331, shoulder=lefty, elbow=epositive, wrist=wpositive, fatherId=fReference[0]}
  [3343] = {x=-615.558, y=233.706, z=44, rx=180, rz=164.501, shoulder=lefty, elbow=epositive, wrist=wpositive, fatherId=fReference[0]}
  [3344] = {x=-614.17, y=234.091, z=44, rx=180, rz=164.672, shoulder=lefty, elbow=epositive, wrist=wpositive, fatherId=fReference[0]}
  [3345] = {x=-612.781, y=234.471, z=44, rx=180, rz=164.843, shoulder=lefty, elbow=epositive, wrist=wpositive, fatherId=fReference[0]}
  [3346] = {x=-611.392, y=234.848, z=44, rx=180, rz=165.015, shoulder=lefty, elbow=epositive, wrist=wpositive, fatherId=fReference[0]}
  [3347] = {x=-610.002, y=235.22, z=44, rx=180, rz=165.188, shoulder=lefty, elbow=epositive, wrist=wpositive, fatherId=fReference[0]}
  [3348] = {x=-608.612, y=235.587, z=44, rx=-180, rz=165.361, shoulder=lefty, elbow=epositive, wrist=wpositive, fatherId=fReference[0]}
  [3349] = {x=-607.221, y=235.951, z=44, rx=180, rz=165.535, shoulder=lefty, elbow=epositive, wrist=wpositive, fatherId=fReference[0]}
  [3350] = {x=-605.829, y=236.31, z=44, rx=180, rz=165.71, shoulder=lefty, elbow=epositive, wrist=wpositive, fatherId=fReference[0]}
  [3351] = {x=-604.437, y=236.664, z=44, rx=180, rz=165.885, shoulder=lefty, elbow=epositive, wrist=wpositive, fatherId=fReference[0]}
  [3352] = {x=-603.045, y=237.014, z=44, rx=180, rz=166.061, shoulder=lefty, elbow=epositive, wrist=wpositive, fatherId=fReference[0]}
  [3353] = {x=-601.652, y=237.36, z=44, rx=180, rz=166.237, shoulder=lefty, elbow=epositive, wrist=wpositive, fatherId=fReference[0]}
  [3354] = {x=-600.258, y=237.701, z=44, rx=180, rz=166.414, shoulder=lefty, elbow=epositive, wrist=wpositive, fatherId=fReference[0]}
  [3355] = {x=-598.864, y=238.038, z=44, rx=180, rz=166.591, shoulder=lefty, elbow=epositive, wrist=wpositive, fatherId=fReference[0]}
  [3356] = {x=-597.469, y=238.371, z=44, rx=180, rz=166.77, shoulder=lefty, elbow=epositive, wrist=wpositive, fatherId=fReference[0]}
  [3357] = {x=-596.074, y=238.699, z=44, rx=180, rz=166.948, shoulder=lefty, elbow=epositive, wrist=wpositive, fatherId=fReference[0]}
  [3358] = {x=-594.678, y=239.023, z=44, rx=180, rz=167.127, shoulder=lefty, elbow=epositive, wrist=wpositive, fatherId=fReference[0]}
  [3359] = {x=-593.281, y=239.342, z=44, rx=180, rz=167.307, shoulder=lefty, elbow=epositive, wrist=wpositive, fatherId=fReference[0]}
  [3360] = {x=-591.885, y=239.656, z=44, rx=180, rz=167.487, shoulder=lefty, elbow=epositive, wrist=wpositive, fatherId=fReference[0]}
  [3361] = {x=-590.487, y=239.966, z=44, rx=180, rz=167.668, shoulder=lefty, elbow=epositive, wrist=wpositive, fatherId=fReference[0]}
  [3362] = {x=-589.09, y=240.272, z=44, rx=180, rz=167.85, shoulder=lefty, elbow=epositive, wrist=wpositive, fatherId=fReference[0]}
  [3363] = {x=-587.691, y=240.573, z=44, rx=180, rz=168.032, shoulder=lefty, elbow=epositive, wrist=wpositive, fatherId=fReference[0]}
  [3364] = {x=-586.292, y=240.869, z=44, rx=180, rz=168.214, shoulder=lefty, elbow=epositive, wrist=wpositive, fatherId=fReference[0]}
  [3365] = {x=-584.893, y=241.161, z=44, rx=-180, rz=168.397, shoulder=lefty, elbow=epositive, wrist=wpositive, fatherId=fReference[0]}
  [3366] = {x=-583.493, y=241.449, z=44, rx=180, rz=168.581, shoulder=lefty, elbow=epositive, wrist=wpositive, fatherId=fReference[0]}
  [3367] = {x=-582.093, y=241.732, z=44, rx=180, rz=168.765, shoulder=lefty, elbow=epositive, wrist=wpositive, fatherId=fReference[0]}
  [3368] = {x=-580.693, y=242.01, z=44, rx=180, rz=168.949, shoulder=lefty, elbow=epositive, wrist=wpositive, fatherId=fReference[0]}
  [3369] = {x=-579.292, y=242.283, z=44, rx=180, rz=169.134, shoulder=lefty, elbow=epositive, wrist=wpositive, fatherId=fReference[0]}
  [3370] = {x=-577.89, y=242.553, z=44, rx=-180, rz=169.32, shoulder=lefty, elbow=epositive, wrist=wpositive, fatherId=fReference[0]}
  [3371] = {x=-576.488, y=242.817, z=44, rx=180, rz=169.506, shoulder=lefty, elbow=epositive, wrist=wpositive, fatherId=fReference[0]}
  [3372] = {x=-575.086, y=243.077, z=44, rx=180, rz=169.692, shoulder=lefty, elbow=epositive, wrist=wpositive, fatherId=fReference[0]}
  [3373] = {x=-573.683, y=243.332, z=44, rx=-180, rz=169.879, shoulder=lefty, elbow=epositive, wrist=wpositive, fatherId=fReference[0]}
  [3374] = {x=-572.279, y=243.582, z=44, rx=-180, rz=170.067, shoulder=lefty, elbow=epositive, wrist=wpositive, fatherId=fReference[0]}
  [3375] = {x=-570.876, y=243.828, z=44, rx=-180, rz=170.255, shoulder=lefty, elbow=epositive, wrist=wpositive, fatherId=fReference[0]}
  [3376] = {x=-569.472, y=244.069, z=44, rx=-180, rz=170.443, shoulder=lefty, elbow=epositive, wrist=wpositive, fatherId=fReference[0]}
  [3377] = {x=-568.067, y=244.306, z=44, rx=180, rz=170.632, shoulder=lefty, elbow=epositive, wrist=wpositive, fatherId=fReference[0]}
  [3378] = {x=-566.662, y=244.538, z=44, rx=-180, rz=170.821, shoulder=lefty, elbow=epositive, wrist=wpositive, fatherId=fReference[0]}
  [3379] = {x=-565.257, y=244.765, z=44, rx=180, rz=171.011, shoulder=lefty, elbow=epositive, wrist=wpositive, fatherId=fReference[0]}
  [3380] = {x=-563.852, y=244.987, z=44, rx=-180, rz=171.201, shoulder=lefty, elbow=epositive, wrist=wpositive, fatherId=fReference[0]}
  [3381] = {x=-562.446, y=245.205, z=44, rx=180, rz=171.391, shoulder=lefty, elbow=epositive, wrist=wpositive, fatherId=fReference[0]}
  [3382] = {x=-561.039, y=245.417, z=44, rx=180, rz=171.582, shoulder=lefty, elbow=epositive, wrist=wpositive, fatherId=fReference[0]}
  [3383] = {x=-559.632, y=245.626, z=44, rx=-180, rz=171.774, shoulder=lefty, elbow=epositive, wrist=wpositive, fatherId=fReference[0]}
  [3384] = {x=-558.225, y=245.829, z=44, rx=-180, rz=171.965, shoulder=lefty, elbow=epositive, wrist=wpositive, fatherId=fReference[0]}
  [3385] = {x=-556.818, y=246.028, z=44, rx=180, rz=172.157, shoulder=lefty, elbow=epositive, wrist=wpositive, fatherId=fReference[0]}
  [3386] = {x=-555.41, y=246.222, z=44, rx=180, rz=172.35, shoulder=lefty, elbow=epositive, wrist=wpositive, fatherId=fReference[0]}
  [3387] = {x=-554.002, y=246.411, z=44, rx=-180, rz=172.543, shoulder=lefty, elbow=epositive, wrist=wpositive, fatherId=fReference[0]}
  [3388] = {x=-552.594, y=246.595, z=44, rx=-180, rz=172.736, shoulder=lefty, elbow=epositive, wrist=wpositive, fatherId=fReference[0]}
  [3389] = {x=-551.185, y=246.775, z=44, rx=180, rz=172.929, shoulder=lefty, elbow=epositive, wrist=wpositive, fatherId=fReference[0]}
  [3390] = {x=-549.776, y=246.949, z=44, rx=180, rz=173.123, shoulder=lefty, elbow=epositive, wrist=wpositive, fatherId=fReference[0]}
  [3391] = {x=-548.367, y=247.119, z=44, rx=180, rz=173.317, shoulder=lefty, elbow=epositive, wrist=wpositive, fatherId=fReference[0]}
  [3392] = {x=-546.957, y=247.285, z=44, rx=180, rz=173.512, shoulder=lefty, elbow=epositive, wrist=wpositive, fatherId=fReference[0]}
  [3393] = {x=-545.548, y=247.445, z=44, rx=180, rz=173.707, shoulder=lefty, elbow=epositive, wrist=wpositive, fatherId=fReference[0]}
  [3394] = {x=-544.137, y=247.6, z=44, rx=-180, rz=173.902, shoulder=lefty, elbow=epositive, wrist=wpositive, fatherId=fReference[0]}
  [3395] = {x=-542.727, y=247.751, z=44, rx=180, rz=174.097, shoulder=lefty, elbow=epositive, wrist=wpositive, fatherId=fReference[0]}
  [3396] = {x=-541.316, y=247.897, z=44, rx=180, rz=174.293, shoulder=lefty, elbow=epositive, wrist=wpositive, fatherId=fReference[0]}
  [3397] = {x=-539.905, y=248.038, z=44, rx=180, rz=174.489, shoulder=lefty, elbow=epositive, wrist=wpositive, fatherId=fReference[0]}
  [3398] = {x=-538.494, y=248.174, z=44, rx=180, rz=174.685, shoulder=lefty, elbow=epositive, wrist=wpositive, fatherId=fReference[0]}
  [3399] = {x=-537.083, y=248.305, z=44, rx=180, rz=174.882, shoulder=lefty, elbow=epositive, wrist=wpositive, fatherId=fReference[0]}
  [3400] = {x=-535.671, y=248.432, z=44, rx=180, rz=175.079, shoulder=lefty, elbow=epositive, wrist=wpositive, fatherId=fReference[0]}
  [3401] = {x=-534.26, y=248.553, z=44, rx=-180, rz=175.276, shoulder=lefty, elbow=epositive, wrist=wpositive, fatherId=fReference[0]}
  [3402] = {x=-532.848, y=248.67, z=44, rx=-180, rz=175.473, shoulder=lefty, elbow=epositive, wrist=wpositive, fatherId=fReference[0]}
  [3403] = {x=-531.435, y=248.782, z=44, rx=180, rz=175.671, shoulder=lefty, elbow=epositive, wrist=wpositive, fatherId=fReference[0]}
  [3404] = {x=-530.023, y=248.889, z=44, rx=180, rz=175.868, shoulder=lefty, elbow=epositive, wrist=wpositive, fatherId=fReference[0]}
  [3405] = {x=-528.61, y=248.991, z=44, rx=-180, rz=176.066, shoulder=lefty, elbow=epositive, wrist=wpositive, fatherId=fReference[0]}
  [3406] = {x=-527.198, y=249.088, z=44, rx=180, rz=176.264, shoulder=lefty, elbow=epositive, wrist=wpositive, fatherId=fReference[0]}
  [3407] = {x=-525.785, y=249.18, z=44, rx=180, rz=176.463, shoulder=lefty, elbow=epositive, wrist=wpositive, fatherId=fReference[0]}
  [3408] = {x=-524.372, y=249.268, z=44, rx=-180, rz=176.661, shoulder=lefty, elbow=epositive, wrist=wpositive, fatherId=fReference[0]}
  [3409] = {x=-522.958, y=249.35, z=44, rx=180, rz=176.86, shoulder=lefty, elbow=epositive, wrist=wpositive, fatherId=fReference[0]}
  [3410] = {x=-521.545, y=249.428, z=44, rx=180, rz=177.059, shoulder=lefty, elbow=epositive, wrist=wpositive, fatherId=fReference[0]}
  [3411] = {x=-520.132, y=249.5, z=44, rx=180, rz=177.258, shoulder=lefty, elbow=epositive, wrist=wpositive, fatherId=fReference[0]}
  [3412] = {x=-518.718, y=249.568, z=44, rx=-180, rz=177.457, shoulder=lefty, elbow=epositive, wrist=wpositive, fatherId=fReference[0]}
  [3413] = {x=-517.304, y=249.631, z=44, rx=-180, rz=177.656, shoulder=lefty, elbow=epositive, wrist=wpositive, fatherId=fReference[0]}
  [3414] = {x=-515.89, y=249.689, z=44, rx=180, rz=177.855, shoulder=lefty, elbow=epositive, wrist=wpositive, fatherId=fReference[0]}
  [3415] = {x=-514.476, y=249.742, z=44, rx=180, rz=178.055, shoulder=lefty, elbow=epositive, wrist=wpositive, fatherId=fReference[0]}
  [3416] = {x=-513.062, y=249.79, z=44, rx=-180, rz=178.254, shoulder=lefty, elbow=epositive, wrist=wpositive, fatherId=fReference[0]}
  [3417] = {x=-511.648, y=249.833, z=44, rx=180, rz=178.454, shoulder=lefty, elbow=epositive, wrist=wpositive, fatherId=fReference[0]}
  [3418] = {x=-510.234, y=249.871, z=44, rx=-180, rz=178.654, shoulder=lefty, elbow=epositive, wrist=wpositive, fatherId=fReference[0]}
  [3419] = {x=-508.82, y=249.904, z=44, rx=180, rz=178.853, shoulder=lefty, elbow=epositive, wrist=wpositive, fatherId=fReference[0]}
  [3420] = {x=-507.405, y=249.932, z=44, rx=180, rz=179.053, shoulder=lefty, elbow=epositive, wrist=wpositive, fatherId=fReference[0]}
  [3421] = {x=-505.991, y=249.956, z=44, rx=-180, rz=179.253, shoulder=lefty, elbow=epositive, wrist=wpositive, fatherId=fReference[0]}
  [3422] = {x=-504.577, y=249.974, z=44, rx=-180, rz=179.453, shoulder=lefty, elbow=epositive, wrist=wpositive, fatherId=fReference[0]}
  [3423] = {x=-503.162, y=249.988, z=44, rx=180, rz=179.653, shoulder=lefty, elbow=epositive, wrist=wpositive, fatherId=fReference[0]}
  [3424] = {x=-501.748, y=249.996, z=44, rx=180, rz=179.853, shoulder=lefty, elbow=epositive, wrist=wpositive, fatherId=fReference[0]}
  [3425] = {x=-500.333, y=250, z=44, rx=180, rz=-179.947, shoulder=lefty, elbow=epositive, wrist=wpositive, fatherId=fReference[0]}
  [3426] = {x=-498.919, y=249.999, z=44, rx=-180, rz=-179.747, shoulder=lefty, elbow=epositive, wrist=wpositive, fatherId=fReference[0]}
  [3427] = {x=-497.504, y=249.992, z=44, rx=-180, rz=-179.547, shoulder=lefty, elbow=epositive, wrist=wpositive, fatherId=fReference[0]}
  [3428] = {x=-496.09, y=249.981, z=44, rx=180, rz=-179.347, shoulder=lefty, elbow=epositive, wrist=wpositive, fatherId=fReference[0]}
  [3429] = {x=-494.676, y=249.965, z=44, rx=180, rz=-179.147, shoulder=lefty, elbow=epositive, wrist=wpositive, fatherId=fReference[0]}
  [3430] = {x=-493.261, y=249.944, z=44, rx=180, rz=-178.947, shoulder=lefty, elbow=epositive, wrist=wpositive, fatherId=fReference[0]}
  [3431] = {x=-491.847, y=249.918, z=44, rx=-180, rz=-178.748, shoulder=lefty, elbow=epositive, wrist=wpositive, fatherId=fReference[0]}
  [3432] = {x=-490.433, y=249.887, z=44, rx=180, rz=-178.548, shoulder=lefty, elbow=epositive, wrist=wpositive, fatherId=fReference[0]}
  [3433] = {x=-489.019, y=249.851, z=44, rx=-180, rz=-178.348, shoulder=lefty, elbow=epositive, wrist=wpositive, fatherId=fReference[0]}
  [3434] = {x=-487.604, y=249.81, z=44, rx=180, rz=-178.149, shoulder=lefty, elbow=epositive, wrist=wpositive, fatherId=fReference[0]}
  [3435] = {x=-486.19, y=249.765, z=44, rx=-180, rz=-177.949, shoulder=lefty, elbow=epositive, wrist=wpositive, fatherId=fReference[0]}
  [3436] = {x=-484.776, y=249.714, z=44, rx=180, rz=-177.75, shoulder=lefty, elbow=epositive, wrist=wpositive, fatherId=fReference[0]}
  [3437] = {x=-483.363, y=249.659, z=44, rx=-180, rz=-177.551, shoulder=lefty, elbow=epositive, wrist=wpositive, fatherId=fReference[0]}
  [3438] = {x=-481.949, y=249.598, z=44, rx=180, rz=-177.351, shoulder=lefty, elbow=epositive, wrist=wpositive, fatherId=fReference[0]}
  [3439] = {x=-480.535, y=249.533, z=44, rx=180, rz=-177.152, shoulder=lefty, elbow=epositive, wrist=wpositive, fatherId=fReference[0]}
  [3440] = {x=-479.122, y=249.462, z=44, rx=180, rz=-176.954, shoulder=lefty, elbow=epositive, wrist=wpositive, fatherId=fReference[0]}
  [3441] = {x=-477.708, y=249.387, z=44, rx=-180, rz=-176.755, shoulder=lefty, elbow=epositive, wrist=wpositive, fatherId=fReference[0]}
  [3442] = {x=-476.295, y=249.307, z=44, rx=180, rz=-176.556, shoulder=lefty, elbow=epositive, wrist=wpositive, fatherId=fReference[0]}
  [3443] = {x=-474.882, y=249.222, z=44, rx=180, rz=-176.358, shoulder=lefty, elbow=epositive, wrist=wpositive, fatherId=fReference[0]}
  [3444] = {x=-473.469, y=249.132, z=44, rx=-180, rz=-176.16, shoulder=lefty, elbow=epositive, wrist=wpositive, fatherId=fReference[0]}
  [3445] = {x=-472.056, y=249.037, z=44, rx=180, rz=-175.962, shoulder=lefty, elbow=epositive, wrist=wpositive, fatherId=fReference[0]}
  [3446] = {x=-470.643, y=248.937, z=44, rx=-180, rz=-175.764, shoulder=lefty, elbow=epositive, wrist=wpositive, fatherId=fReference[0]}
  [3447] = {x=-469.231, y=248.833, z=44, rx=180, rz=-175.566, shoulder=lefty, elbow=epositive, wrist=wpositive, fatherId=fReference[0]}
  [3448] = {x=-467.819, y=248.723, z=44, rx=-180, rz=-175.369, shoulder=lefty, elbow=epositive, wrist=wpositive, fatherId=fReference[0]}
  [3449] = {x=-466.407, y=248.609, z=44, rx=180, rz=-175.172, shoulder=lefty, elbow=epositive, wrist=wpositive, fatherId=fReference[0]}
  [3450] = {x=-464.995, y=248.49, z=44, rx=180, rz=-174.975, shoulder=lefty, elbow=epositive, wrist=wpositive, fatherId=fReference[0]}
  [3451] = {x=-463.583, y=248.366, z=44, rx=180, rz=-174.778, shoulder=lefty, elbow=epositive, wrist=wpositive, fatherId=fReference[0]}
  [3452] = {x=-462.172, y=248.237, z=44, rx=-180, rz=-174.582, shoulder=lefty, elbow=epositive, wrist=wpositive, fatherId=fReference[0]}
  [3453] = {x=-460.76, y=248.103, z=44, rx=180, rz=-174.386, shoulder=lefty, elbow=epositive, wrist=wpositive, fatherId=fReference[0]}
  [3454] = {x=-459.349, y=247.964, z=44, rx=180, rz=-174.19, shoulder=lefty, elbow=epositive, wrist=wpositive, fatherId=fReference[0]}
  [3455] = {x=-457.939, y=247.82, z=44, rx=180, rz=-173.994, shoulder=lefty, elbow=epositive, wrist=wpositive, fatherId=fReference[0]}
  [3456] = {x=-456.528, y=247.672, z=44, rx=180, rz=-173.799, shoulder=lefty, elbow=epositive, wrist=wpositive, fatherId=fReference[0]}
  [3457] = {x=-455.118, y=247.519, z=44, rx=-180, rz=-173.604, shoulder=lefty, elbow=epositive, wrist=wpositive, fatherId=fReference[0]}
  [3458] = {x=-453.708, y=247.361, z=44, rx=-180, rz=-173.409, shoulder=lefty, elbow=epositive, wrist=wpositive, fatherId=fReference[0]}
  [3459] = {x=-452.298, y=247.198, z=44, rx=-180, rz=-173.215, shoulder=lefty, elbow=epositive, wrist=wpositive, fatherId=fReference[0]}
  [3460] = {x=-450.889, y=247.03, z=44, rx=180, rz=-173.021, shoulder=lefty, elbow=epositive, wrist=wpositive, fatherId=fReference[0]}
  [3461] = {x=-449.48, y=246.858, z=44, rx=180, rz=-172.827, shoulder=lefty, elbow=epositive, wrist=wpositive, fatherId=fReference[0]}
  [3462] = {x=-448.071, y=246.68, z=44, rx=-180, rz=-172.634, shoulder=lefty, elbow=epositive, wrist=wpositive, fatherId=fReference[0]}
  [3463] = {x=-446.663, y=246.498, z=44, rx=180, rz=-172.441, shoulder=lefty, elbow=epositive, wrist=wpositive, fatherId=fReference[0]}
  [3464] = {x=-445.254, y=246.312, z=44, rx=180, rz=-172.248, shoulder=lefty, elbow=epositive, wrist=wpositive, fatherId=fReference[0]}
  [3465] = {x=-443.847, y=246.12, z=44, rx=180, rz=-172.056, shoulder=lefty, elbow=epositive, wrist=wpositive, fatherId=fReference[0]}
  [3466] = {x=-442.439, y=245.923, z=44, rx=-180, rz=-171.864, shoulder=lefty, elbow=epositive, wrist=wpositive, fatherId=fReference[0]}
  [3467] = {x=-441.032, y=245.722, z=44, rx=180, rz=-171.673, shoulder=lefty, elbow=epositive, wrist=wpositive, fatherId=fReference[0]}
  [3468] = {x=-439.625, y=245.516, z=44, rx=180, rz=-171.482, shoulder=lefty, elbow=epositive, wrist=wpositive, fatherId=fReference[0]}
  [3469] = {x=-438.218, y=245.306, z=44, rx=-180, rz=-171.291, shoulder=lefty, elbow=epositive, wrist=wpositive, fatherId=fReference[0]}
  [3470] = {x=-436.812, y=245.09, z=44, rx=-180, rz=-171.101, shoulder=lefty, elbow=epositive, wrist=wpositive, fatherId=fReference[0]}
  [3471] = {x=-435.406, y=244.87, z=44, rx=-180, rz=-170.911, shoulder=lefty, elbow=epositive, wrist=wpositive, fatherId=fReference[0]}
  [3472] = {x=-434.001, y=244.645, z=44, rx=-180, rz=-170.721, shoulder=lefty, elbow=epositive, wrist=wpositive, fatherId=fReference[0]}
  [3473] = {x=-432.596, y=244.416, z=44, rx=-180, rz=-170.532, shoulder=lefty, elbow=epositive, wrist=wpositive, fatherId=fReference[0]}
  [3474] = {x=-431.191, y=244.182, z=44, rx=-180, rz=-170.344, shoulder=lefty, elbow=epositive, wrist=wpositive, fatherId=fReference[0]}
  [3475] = {x=-429.787, y=243.943, z=44, rx=180, rz=-170.156, shoulder=lefty, elbow=epositive, wrist=wpositive, fatherId=fReference[0]}
  [3476] = {x=-428.383, y=243.699, z=44, rx=180, rz=-169.968, shoulder=lefty, elbow=epositive, wrist=wpositive, fatherId=fReference[0]}
  [3477] = {x=-426.98, y=243.451, z=44, rx=180, rz=-169.781, shoulder=lefty, elbow=epositive, wrist=wpositive, fatherId=fReference[0]}
  [3478] = {x=-425.577, y=243.198, z=44, rx=-180, rz=-169.594, shoulder=lefty, elbow=epositive, wrist=wpositive, fatherId=fReference[0]}
  [3479] = {x=-424.174, y=242.94, z=44, rx=-180, rz=-169.408, shoulder=lefty, elbow=epositive, wrist=wpositive, fatherId=fReference[0]}
  [3480] = {x=-422.772, y=242.678, z=44, rx=180, rz=-169.222, shoulder=lefty, elbow=epositive, wrist=wpositive, fatherId=fReference[0]}
  [3481] = {x=-421.37, y=242.411, z=44, rx=180, rz=-169.037, shoulder=lefty, elbow=epositive, wrist=wpositive, fatherId=fReference[0]}
  [3482] = {x=-419.969, y=242.14, z=44, rx=-180, rz=-168.852, shoulder=lefty, elbow=epositive, wrist=wpositive, fatherId=fReference[0]}
  [3483] = {x=-418.568, y=241.864, z=44, rx=-180, rz=-168.667, shoulder=lefty, elbow=epositive, wrist=wpositive, fatherId=fReference[0]}
  [3484] = {x=-417.167, y=241.583, z=44, rx=180, rz=-168.484, shoulder=lefty, elbow=epositive, wrist=wpositive, fatherId=fReference[0]}
  [3485] = {x=-415.767, y=241.298, z=44, rx=-180, rz=-168.3, shoulder=lefty, elbow=epositive, wrist=wpositive, fatherId=fReference[0]}
  [3486] = {x=-414.368, y=241.008, z=44, rx=-180, rz=-168.118, shoulder=lefty, elbow=epositive, wrist=wpositive, fatherId=fReference[0]}
  [3487] = {x=-412.969, y=240.713, z=44, rx=180, rz=-167.935, shoulder=lefty, elbow=epositive, wrist=wpositive, fatherId=fReference[0]}
  [3488] = {x=-411.57, y=240.415, z=44, rx=180, rz=-167.754, shoulder=lefty, elbow=epositive, wrist=wpositive, fatherId=fReference[0]}
  [3489] = {x=-410.172, y=240.111, z=44, rx=-180, rz=-167.573, shoulder=lefty, elbow=epositive, wrist=wpositive, fatherId=fReference[0]}
  [3490] = {x=-408.775, y=239.803, z=44, rx=180, rz=-167.392, shoulder=lefty, elbow=epositive, wrist=wpositive, fatherId=fReference[0]}
  [3491] = {x=-407.378, y=239.491, z=44, rx=180, rz=-167.212, shoulder=lefty, elbow=epositive, wrist=wpositive, fatherId=fReference[0]}
  [3492] = {x=-405.981, y=239.174, z=44, rx=-180, rz=-167.033, shoulder=lefty, elbow=epositive, wrist=wpositive, fatherId=fReference[0]}
  [3493] = {x=-404.585, y=238.852, z=44, rx=-180, rz=-166.854, shoulder=lefty, elbow=epositive, wrist=wpositive, fatherId=fReference[0]}
  [3494] = {x=-403.189, y=238.526, z=44, rx=180, rz=-166.675, shoulder=lefty, elbow=epositive, wrist=wpositive, fatherId=fReference[0]}
  [3495] = {x=-401.794, y=238.196, z=44, rx=-180, rz=-166.498, shoulder=lefty, elbow=epositive, wrist=wpositive, fatherId=fReference[0]}
  [3496] = {x=-400.4, y=237.861, z=44, rx=-180, rz=-166.32, shoulder=lefty, elbow=epositive, wrist=wpositive, fatherId=fReference[0]}
  [3497] = {x=-399.006, y=237.522, z=44, rx=180, rz=-166.144, shoulder=lefty, elbow=epositive, wrist=wpositive, fatherId=fReference[0]}
  [3498] = {x=-397.613, y=237.178, z=44, rx=-180, rz=-165.968, shoulder=lefty, elbow=epositive, wrist=wpositive, fatherId=fReference[0]}
  [3499] = {x=-396.22, y=236.83, z=44, rx=180, rz=-165.792, shoulder=lefty, elbow=epositive, wrist=wpositive, fatherId=fReference[0]}
  [3500] = {x=-394.827, y=236.477, z=44, rx=180, rz=-165.618, shoulder=lefty, elbow=epositive, wrist=wpositive, fatherId=fReference[0]}
  [3501] = {x=-393.436, y=236.12, z=44, rx=180, rz=-165.443, shoulder=lefty, elbow=epositive, wrist=wpositive, fatherId=fReference[0]}
  [3502] = {x=-392.044, y=235.759, z=44, rx=-180, rz=-165.27, shoulder=lefty, elbow=epositive, wrist=wpositive, fatherId=fReference[0]}
  [3503] = {x=-390.654, y=235.394, z=44, rx=-180, rz=-165.097, shoulder=lefty, elbow=epositive, wrist=wpositive, fatherId=fReference[0]}
  [3504] = {x=-389.264, y=235.024, z=44, rx=-180, rz=-164.924, shoulder=lefty, elbow=epositive, wrist=wpositive, fatherId=fReference[0]}
  [3505] = {x=-387.874, y=234.649, z=44, rx=-180, rz=-164.753, shoulder=lefty, elbow=epositive, wrist=wpositive, fatherId=fReference[0]}
  [3506] = {x=-386.485, y=234.271, z=44, rx=-180, rz=-164.582, shoulder=lefty, elbow=epositive, wrist=wpositive, fatherId=fReference[0]}
  [3507] = {x=-385.097, y=233.888, z=44, rx=-180, rz=-164.411, shoulder=lefty, elbow=epositive, wrist=wpositive, fatherId=fReference[0]}
  [3508] = {x=-383.709, y=233.501, z=44, rx=-180, rz=-164.241, shoulder=lefty, elbow=epositive, wrist=wpositive, fatherId=fReference[0]}
  [3509] = {x=-382.322, y=233.109, z=44, rx=180, rz=-164.072, shoulder=lefty, elbow=epositive, wrist=wpositive, fatherId=fReference[0]}
  [3510] = {x=-380.936, y=232.714, z=44, rx=-180, rz=-163.904, shoulder=lefty, elbow=epositive, wrist=wpositive, fatherId=fReference[0]}
  [3511] = {x=-379.55, y=232.314, z=44, rx=180, rz=-163.736, shoulder=lefty, elbow=epositive, wrist=wpositive, fatherId=fReference[0]}
  [3512] = {x=-378.164, y=231.909, z=44, rx=180, rz=-163.568, shoulder=lefty, elbow=epositive, wrist=wpositive, fatherId=fReference[0]}
  [3513] = {x=-376.78, y=231.501, z=44, rx=180, rz=-163.402, shoulder=lefty, elbow=epositive, wrist=wpositive, fatherId=fReference[0]}
  [3514] = {x=-375.395, y=231.089, z=44, rx=180, rz=-163.236, shoulder=lefty, elbow=epositive, wrist=wpositive, fatherId=fReference[0]}
  [3515] = {x=-374.012, y=230.672, z=44, rx=180, rz=-163.071, shoulder=lefty, elbow=epositive, wrist=wpositive, fatherId=fReference[0]}
  [3516] = {x=-372.629, y=230.251, z=44, rx=180, rz=-162.906, shoulder=lefty, elbow=epositive, wrist=wpositive, fatherId=fReference[0]}
  [3517] = {x=-371.247, y=229.826, z=44, rx=-180, rz=-162.742, shoulder=lefty, elbow=epositive, wrist=wpositive, fatherId=fReference[0]}
  [3518] = {x=-369.865, y=229.397, z=44, rx=-180, rz=-162.579, shoulder=lefty, elbow=epositive, wrist=wpositive, fatherId=fReference[0]}
  [3519] = {x=-368.484, y=228.963, z=44, rx=-180, rz=-162.416, shoulder=lefty, elbow=epositive, wrist=wpositive, fatherId=fReference[0]}
  [3520] = {x=-367.104, y=228.526, z=44, rx=180, rz=-162.254, shoulder=lefty, elbow=epositive, wrist=wpositive, fatherId=fReference[0]}
  [3521] = {x=-365.724, y=228.084, z=44, rx=180, rz=-162.093, shoulder=lefty, elbow=epositive, wrist=wpositive, fatherId=fReference[0]}
  [3522] = {x=-364.345, y=227.639, z=44, rx=-180, rz=-161.932, shoulder=lefty, elbow=epositive, wrist=wpositive, fatherId=fReference[0]}
  [3523] = {x=-362.966, y=227.189, z=44, rx=-180, rz=-161.772, shoulder=lefty, elbow=epositive, wrist=wpositive, fatherId=fReference[0]}
  [3524] = {x=-361.588, y=226.735, z=44, rx=-180, rz=-161.613, shoulder=lefty, elbow=epositive, wrist=wpositive, fatherId=fReference[0]}
  [3525] = {x=-360.211, y=226.277, z=44, rx=180, rz=-161.455, shoulder=lefty, elbow=epositive, wrist=wpositive, fatherId=fReference[0]}
  [3526] = {x=-358.835, y=225.816, z=44, rx=180, rz=-161.297, shoulder=lefty, elbow=epositive, wrist=wpositive, fatherId=fReference[0]}
  [3527] = {x=-357.459, y=225.35, z=44, rx=180, rz=-161.14, shoulder=lefty, elbow=epositive, wrist=wpositive, fatherId=fReference[0]}
  [3528] = {x=-356.084, y=224.88, z=44, rx=-180, rz=-160.983, shoulder=lefty, elbow=epositive, wrist=wpositive, fatherId=fReference[0]}
  [3529] = {x=-354.709, y=224.406, z=44, rx=-180, rz=-160.828, shoulder=lefty, elbow=epositive, wrist=wpositive, fatherId=fReference[0]}
  [3530] = {x=-353.335, y=223.929, z=44, rx=-180, rz=-160.673, shoulder=lefty, elbow=epositive, wrist=wpositive, fatherId=fReference[0]}
  [3531] = {x=-351.962, y=223.447, z=44, rx=180, rz=-160.518, shoulder=lefty, elbow=epositive, wrist=wpositive, fatherId=fReference[0]}
  [3532] = {x=-350.59, y=222.961, z=44, rx=-180, rz=-160.365, shoulder=lefty, elbow=epositive, wrist=wpositive, fatherId=fReference[0]}
  [3533] = {x=-349.218, y=222.472, z=44, rx=-180, rz=-160.212, shoulder=lefty, elbow=epositive, wrist=wpositive, fatherId=fReference[0]}
  [3534] = {x=-347.847, y=221.979, z=44, rx=180, rz=-160.06, shoulder=lefty, elbow=epositive, wrist=wpositive, fatherId=fReference[0]}
  [3535] = {x=-346.476, y=221.482, z=44, rx=180, rz=-159.908, shoulder=lefty, elbow=epositive, wrist=wpositive, fatherId=fReference[0]}
  [3536] = {x=-345.107, y=220.98, z=44, rx=-180, rz=-159.757, shoulder=lefty, elbow=epositive, wrist=wpositive, fatherId=fReference[0]}
  [3537] = {x=-343.737, y=220.476, z=44, rx=180, rz=-159.607, shoulder=lefty, elbow=epositive, wrist=wpositive, fatherId=fReference[0]}
  [3538] = {x=-342.369, y=219.967, z=44, rx=180, rz=-159.458, shoulder=lefty, elbow=epositive, wrist=wpositive, fatherId=fReference[0]}
  [3539] = {x=-341.001, y=219.454, z=44, rx=-180, rz=-159.309, shoulder=lefty, elbow=epositive, wrist=wpositive, fatherId=fReference[0]}
  [3540] = {x=-339.634, y=218.938, z=44, rx=-180, rz=-159.161, shoulder=lefty, elbow=epositive, wrist=wpositive, fatherId=fReference[0]}
  [3541] = {x=-338.268, y=218.418, z=44, rx=180, rz=-159.014, shoulder=lefty, elbow=epositive, wrist=wpositive, fatherId=fReference[0]}
  [3542] = {x=-336.903, y=217.894, z=44, rx=180, rz=-158.868, shoulder=lefty, elbow=epositive, wrist=wpositive, fatherId=fReference[0]}
  [3543] = {x=-335.538, y=217.367, z=44, rx=180, rz=-158.722, shoulder=lefty, elbow=epositive, wrist=wpositive, fatherId=fReference[0]}
  [3544] = {x=-334.173, y=216.835, z=44, rx=-180, rz=-158.577, shoulder=lefty, elbow=epositive, wrist=wpositive, fatherId=fReference[0]}
  [3545] = {x=-332.81, y=216.3, z=44, rx=180, rz=-158.433, shoulder=lefty, elbow=epositive, wrist=wpositive, fatherId=fReference[0]}
  [3546] = {x=-331.447, y=215.762, z=44, rx=-180, rz=-158.289, shoulder=lefty, elbow=epositive, wrist=wpositive, fatherId=fReference[0]}
  [3547] = {x=-330.085, y=215.219, z=44, rx=-180, rz=-158.146, shoulder=lefty, elbow=epositive, wrist=wpositive, fatherId=fReference[0]}
  [3548] = {x=-328.724, y=214.674, z=44, rx=-180, rz=-158.004, shoulder=lefty, elbow=epositive, wrist=wpositive, fatherId=fReference[0]}
  [3549] = {x=-327.363, y=214.124, z=44, rx=-180, rz=-157.862, shoulder=lefty, elbow=epositive, wrist=wpositive, fatherId=fReference[0]}
  [3550] = {x=-326.004, y=213.571, z=44, rx=-180, rz=-157.722, shoulder=lefty, elbow=epositive, wrist=wpositive, fatherId=fReference[0]}
  [3551] = {x=-324.644, y=213.014, z=44, rx=180, rz=-157.582, shoulder=lefty, elbow=epositive, wrist=wpositive, fatherId=fReference[0]}
  [3552] = {x=-323.286, y=212.453, z=44, rx=180, rz=-157.442, shoulder=lefty, elbow=epositive, wrist=wpositive, fatherId=fReference[0]}
  [3553] = {x=-321.928, y=211.89, z=44, rx=-180, rz=-157.304, shoulder=lefty, elbow=epositive, wrist=wpositive, fatherId=fReference[0]}
  [3554] = {x=-320.571, y=211.322, z=44, rx=-180, rz=-157.166, shoulder=lefty, elbow=epositive, wrist=wpositive, fatherId=fReference[0]}
  [3555] = {x=-319.215, y=210.751, z=44, rx=180, rz=-157.029, shoulder=lefty, elbow=epositive, wrist=wpositive, fatherId=fReference[0]}
  [3556] = {x=-317.86, y=210.176, z=44, rx=-180, rz=-156.893, shoulder=lefty, elbow=epositive, wrist=wpositive, fatherId=fReference[0]}
  [3557] = {x=-316.505, y=209.598, z=44, rx=180, rz=-156.757, shoulder=lefty, elbow=epositive, wrist=wpositive, fatherId=fReference[0]}
  [3558] = {x=-315.151, y=209.017, z=44, rx=-180, rz=-156.622, shoulder=lefty, elbow=epositive, wrist=wpositive, fatherId=fReference[0]}
  [3559] = {x=-313.798, y=208.432, z=44, rx=180, rz=-156.488, shoulder=lefty, elbow=epositive, wrist=wpositive, fatherId=fReference[0]}
  [3560] = {x=-312.445, y=207.843, z=44, rx=-180, rz=-156.354, shoulder=lefty, elbow=epositive, wrist=wpositive, fatherId=fReference[0]}
  [3561] = {x=-311.094, y=207.252, z=44, rx=180, rz=-156.222, shoulder=lefty, elbow=epositive, wrist=wpositive, fatherId=fReference[0]}
  [3562] = {x=-309.743, y=206.656, z=44, rx=-180, rz=-156.09, shoulder=lefty, elbow=epositive, wrist=wpositive, fatherId=fReference[0]}
  [3563] = {x=-308.392, y=206.058, z=44, rx=180, rz=-155.958, shoulder=lefty, elbow=epositive, wrist=wpositive, fatherId=fReference[0]}
  [3564] = {x=-307.043, y=205.456, z=44, rx=-180, rz=-155.828, shoulder=lefty, elbow=epositive, wrist=wpositive, fatherId=fReference[0]}
  [3565] = {x=-305.694, y=204.85, z=44, rx=-180, rz=-155.698, shoulder=lefty, elbow=epositive, wrist=wpositive, fatherId=fReference[0]}
  [3566] = {x=-304.346, y=204.242, z=44, rx=-180, rz=-155.569, shoulder=lefty, elbow=epositive, wrist=wpositive, fatherId=fReference[0]}
  [3567] = {x=-302.999, y=203.63, z=44, rx=180, rz=-155.44, shoulder=lefty, elbow=epositive, wrist=wpositive, fatherId=fReference[0]}
  [3568] = {x=-301.652, y=203.014, z=44, rx=180, rz=-155.312, shoulder=lefty, elbow=epositive, wrist=wpositive, fatherId=fReference[0]}
  [3569] = {x=-300.307, y=202.396, z=44, rx=-180, rz=-155.185, shoulder=lefty, elbow=epositive, wrist=wpositive, fatherId=fReference[0]}
  [3570] = {x=-298.962, y=201.774, z=44, rx=180, rz=-155.059, shoulder=lefty, elbow=epositive, wrist=wpositive, fatherId=fReference[0]}
  [3571] = {x=-297.618, y=201.149, z=44, rx=-180, rz=-154.934, shoulder=lefty, elbow=epositive, wrist=wpositive, fatherId=fReference[0]}
  [3572] = {x=-296.274, y=200.52, z=44, rx=-180, rz=-154.809, shoulder=lefty, elbow=epositive, wrist=wpositive, fatherId=fReference[0]}
  [3573] = {x=-294.931, y=199.889, z=44, rx=180, rz=-154.685, shoulder=lefty, elbow=epositive, wrist=wpositive, fatherId=fReference[0]}
  [3574] = {x=-293.589, y=199.254, z=44, rx=-180, rz=-154.561, shoulder=lefty, elbow=epositive, wrist=wpositive, fatherId=fReference[0]}
  [3575] = {x=-292.248, y=198.616, z=44, rx=-180, rz=-154.439, shoulder=lefty, elbow=epositive, wrist=wpositive, fatherId=fReference[0]}
  [3576] = {x=-290.908, y=197.975, z=44, rx=180, rz=-154.317, shoulder=lefty, elbow=epositive, wrist=wpositive, fatherId=fReference[0]}
  [3577] = {x=-289.568, y=197.331, z=44, rx=-180, rz=-154.195, shoulder=lefty, elbow=epositive, wrist=wpositive, fatherId=fReference[0]}
  [3578] = {x=-288.229, y=196.683, z=44, rx=-180, rz=-154.075, shoulder=lefty, elbow=epositive, wrist=wpositive, fatherId=fReference[0]}
  [3579] = {x=-286.891, y=196.033, z=44, rx=-180, rz=-153.955, shoulder=lefty, elbow=epositive, wrist=wpositive, fatherId=fReference[0]}
  [3580] = {x=-285.554, y=195.379, z=44, rx=-180, rz=-153.836, shoulder=lefty, elbow=epositive, wrist=wpositive, fatherId=fReference[0]}
  [3581] = {x=-284.217, y=194.723, z=44, rx=180, rz=-153.718, shoulder=lefty, elbow=epositive, wrist=wpositive, fatherId=fReference[0]}
  [3582] = {x=-282.882, y=194.063, z=44, rx=180, rz=-153.6, shoulder=lefty, elbow=epositive, wrist=wpositive, fatherId=fReference[0]}
  [3583] = {x=-281.546, y=193.4, z=44, rx=-180, rz=-153.483, shoulder=lefty, elbow=epositive, wrist=wpositive, fatherId=fReference[0]}
  [3584] = {x=-280.212, y=192.734, z=44, rx=-180, rz=-153.367, shoulder=lefty, elbow=epositive, wrist=wpositive, fatherId=fReference[0]}
  [3585] = {x=-278.879, y=192.066, z=44, rx=-180, rz=-153.251, shoulder=lefty, elbow=epositive, wrist=wpositive, fatherId=fReference[0]}
  [3586] = {x=-277.546, y=191.394, z=44, rx=-180, rz=-153.136, shoulder=lefty, elbow=epositive, wrist=wpositive, fatherId=fReference[0]}
  [3587] = {x=-276.214, y=190.719, z=44, rx=180, rz=-153.022, shoulder=lefty, elbow=epositive, wrist=wpositive, fatherId=fReference[0]}
  [3588] = {x=-274.883, y=190.042, z=44, rx=180, rz=-152.908, shoulder=lefty, elbow=epositive, wrist=wpositive, fatherId=fReference[0]}
  [3589] = {x=-273.552, y=189.361, z=44, rx=-180, rz=-152.796, shoulder=lefty, elbow=epositive, wrist=wpositive, fatherId=fReference[0]}
  [3590] = {x=-272.222, y=188.678, z=44, rx=180, rz=-152.684, shoulder=lefty, elbow=epositive, wrist=wpositive, fatherId=fReference[0]}
  [3591] = {x=-270.894, y=187.991, z=44, rx=-180, rz=-152.572, shoulder=lefty, elbow=epositive, wrist=wpositive, fatherId=fReference[0]}
  [3592] = {x=-269.565, y=187.302, z=44, rx=-180, rz=-152.461, shoulder=lefty, elbow=epositive, wrist=wpositive, fatherId=fReference[0]}
  [3593] = {x=-268.238, y=186.61, z=44, rx=180, rz=-152.351, shoulder=lefty, elbow=epositive, wrist=wpositive, fatherId=fReference[0]}
  [3594] = {x=-266.911, y=185.915, z=44, rx=180, rz=-152.242, shoulder=lefty, elbow=epositive, wrist=wpositive, fatherId=fReference[0]}
  [3595] = {x=-265.585, y=185.217, z=44, rx=180, rz=-152.134, shoulder=lefty, elbow=epositive, wrist=wpositive, fatherId=fReference[0]}
  [3596] = {x=-264.26, y=184.516, z=44, rx=180, rz=-152.026, shoulder=lefty, elbow=epositive, wrist=wpositive, fatherId=fReference[0]}
  [3597] = {x=-262.936, y=183.813, z=44, rx=180, rz=-151.918, shoulder=lefty, elbow=epositive, wrist=wpositive, fatherId=fReference[0]}
  [3598] = {x=-261.612, y=183.107, z=44, rx=180, rz=-151.812, shoulder=lefty, elbow=epositive, wrist=wpositive, fatherId=fReference[0]}
  [3599] = {x=-260.289, y=182.398, z=44, rx=-180, rz=-151.706, shoulder=lefty, elbow=epositive, wrist=wpositive, fatherId=fReference[0]}
  [3600] = {x=-258.967, y=181.686, z=44, rx=180, rz=-151.601, shoulder=lefty, elbow=epositive, wrist=wpositive, fatherId=fReference[0]}
  [3601] = {x=-257.646, y=180.972, z=44, rx=-180, rz=-151.496, shoulder=lefty, elbow=epositive, wrist=wpositive, fatherId=fReference[0]}
  [3602] = {x=-256.325, y=180.254, z=44, rx=180, rz=-151.392, shoulder=lefty, elbow=epositive, wrist=wpositive, fatherId=fReference[0]}
  [3603] = {x=-255.005, y=179.535, z=44, rx=180, rz=-151.289, shoulder=lefty, elbow=epositive, wrist=wpositive, fatherId=fReference[0]}
  [3604] = {x=-253.686, y=178.812, z=44, rx=-180, rz=-151.187, shoulder=lefty, elbow=epositive, wrist=wpositive, fatherId=fReference[0]}
  [3605] = {x=-252.368, y=178.087, z=44, rx=180, rz=-151.085, shoulder=lefty, elbow=epositive, wrist=wpositive, fatherId=fReference[0]}
  [3606] = {x=-251.05, y=177.359, z=44, rx=-180, rz=-150.984, shoulder=lefty, elbow=epositive, wrist=wpositive, fatherId=fReference[0]}
  [3607] = {x=-249.733, y=176.629, z=44, rx=-180, rz=-150.883, shoulder=lefty, elbow=epositive, wrist=wpositive, fatherId=fReference[0]}
  [3608] = {x=-248.417, y=175.895, z=44, rx=180, rz=-150.784, shoulder=lefty, elbow=epositive, wrist=wpositive, fatherId=fReference[0]}
  [3609] = {x=-247.102, y=175.16, z=44, rx=-180, rz=-150.685, shoulder=lefty, elbow=epositive, wrist=wpositive, fatherId=fReference[0]}
  [3610] = {x=-245.787, y=174.422, z=44, rx=-180, rz=-150.586, shoulder=lefty, elbow=epositive, wrist=wpositive, fatherId=fReference[0]}
  [3611] = {x=-244.473, y=173.681, z=44, rx=180, rz=-150.488, shoulder=lefty, elbow=epositive, wrist=wpositive, fatherId=fReference[0]}
  [3612] = {x=-243.16, y=172.937, z=44, rx=-180, rz=-150.391, shoulder=lefty, elbow=epositive, wrist=wpositive, fatherId=fReference[0]}
  [3613] = {x=-241.847, y=172.192, z=44, rx=-180, rz=-150.295, shoulder=lefty, elbow=epositive, wrist=wpositive, fatherId=fReference[0]}
  [3614] = {x=-240.536, y=171.443, z=44, rx=180, rz=-150.199, shoulder=lefty, elbow=epositive, wrist=wpositive, fatherId=fReference[0]}
  [3615] = {x=-239.225, y=170.692, z=44, rx=180, rz=-150.104, shoulder=lefty, elbow=epositive, wrist=wpositive, fatherId=fReference[0]}
  [3616] = {x=-237.914, y=169.939, z=44, rx=180, rz=-150.009, shoulder=lefty, elbow=epositive, wrist=wpositive, fatherId=fReference[0]}
  [3617] = {x=-236.605, y=169.183, z=44, rx=-180, rz=-149.915, shoulder=lefty, elbow=epositive, wrist=wpositive, fatherId=fReference[0]}
  [3618] = {x=-235.296, y=168.425, z=44, rx=-180, rz=-149.822, shoulder=lefty, elbow=epositive, wrist=wpositive, fatherId=fReference[0]}
  [3619] = {x=-233.988, y=167.664, z=44, rx=180, rz=-149.729, shoulder=lefty, elbow=epositive, wrist=wpositive, fatherId=fReference[0]}
  [3620] = {x=-232.68, y=166.901, z=44, rx=-180, rz=-149.638, shoulder=lefty, elbow=epositive, wrist=wpositive, fatherId=fReference[0]}
  [3621] = {x=-231.373, y=166.136, z=44, rx=-180, rz=-149.546, shoulder=lefty, elbow=epositive, wrist=wpositive, fatherId=fReference[0]}
  [3622] = {x=-230.067, y=165.368, z=44, rx=-180, rz=-149.456, shoulder=lefty, elbow=epositive, wrist=wpositive, fatherId=fReference[0]}
  [3623] = {x=-228.762, y=164.597, z=44, rx=-180, rz=-149.366, shoulder=lefty, elbow=epositive, wrist=wpositive, fatherId=fReference[0]}
  [3624] = {x=-227.457, y=163.825, z=44, rx=-180, rz=-149.276, shoulder=lefty, elbow=epositive, wrist=wpositive, fatherId=fReference[0]}
  [3625] = {x=-226.153, y=163.05, z=44, rx=-180, rz=-149.187, shoulder=lefty, elbow=epositive, wrist=wpositive, fatherId=fReference[0]}
  [3626] = {x=-224.85, y=162.272, z=44, rx=-180, rz=-149.099, shoulder=lefty, elbow=epositive, wrist=wpositive, fatherId=fReference[0]}
  [3627] = {x=-223.547, y=161.493, z=44, rx=-180, rz=-149.012, shoulder=lefty, elbow=epositive, wrist=wpositive, fatherId=fReference[0]}
  [3628] = {x=-222.245, y=160.711, z=44, rx=180, rz=-148.925, shoulder=lefty, elbow=epositive, wrist=wpositive, fatherId=fReference[0]}
  [3629] = {x=-220.944, y=159.927, z=44, rx=-180, rz=-148.839, shoulder=lefty, elbow=epositive, wrist=wpositive, fatherId=fReference[0]}
  [3630] = {x=-219.643, y=159.14, z=44, rx=-180, rz=-148.753, shoulder=lefty, elbow=epositive, wrist=wpositive, fatherId=fReference[0]}
  [3631] = {x=-218.344, y=158.351, z=44, rx=180, rz=-148.668, shoulder=lefty, elbow=epositive, wrist=wpositive, fatherId=fReference[0]}
  [3632] = {x=-217.044, y=157.56, z=44, rx=180, rz=-148.584, shoulder=lefty, elbow=epositive, wrist=wpositive, fatherId=fReference[0]}
  [3633] = {x=-215.746, y=156.767, z=44, rx=180, rz=-148.5, shoulder=lefty, elbow=epositive, wrist=wpositive, fatherId=fReference[0]}
  [3634] = {x=-214.448, y=155.972, z=44, rx=-180, rz=-148.417, shoulder=lefty, elbow=epositive, wrist=wpositive, fatherId=fReference[0]}
  [3635] = {x=-213.15, y=155.174, z=44, rx=-180, rz=-148.334, shoulder=lefty, elbow=epositive, wrist=wpositive, fatherId=fReference[0]}
  [3636] = {x=-211.854, y=154.375, z=44, rx=-180, rz=-148.252, shoulder=lefty, elbow=epositive, wrist=wpositive, fatherId=fReference[0]}
  [3637] = {x=-210.558, y=153.573, z=44, rx=-180, rz=-148.171, shoulder=lefty, elbow=epositive, wrist=wpositive, fatherId=fReference[0]}
  [3638] = {x=-209.262, y=152.769, z=44, rx=180, rz=-148.09, shoulder=lefty, elbow=epositive, wrist=wpositive, fatherId=fReference[0]}
  [3639] = {x=-207.968, y=151.962, z=44, rx=-180, rz=-148.01, shoulder=lefty, elbow=epositive, wrist=wpositive, fatherId=fReference[0]}
  [3640] = {x=-206.674, y=151.154, z=44, rx=-180, rz=-147.931, shoulder=lefty, elbow=epositive, wrist=wpositive, fatherId=fReference[0]}
  [3641] = {x=-205.38, y=150.344, z=44, rx=180, rz=-147.852, shoulder=lefty, elbow=epositive, wrist=wpositive, fatherId=fReference[0]}
  [3642] = {x=-204.088, y=149.531, z=44, rx=-180, rz=-147.774, shoulder=lefty, elbow=epositive, wrist=wpositive, fatherId=fReference[0]}
  [3643] = {x=-202.795, y=148.717, z=44, rx=180, rz=-147.696, shoulder=lefty, elbow=epositive, wrist=wpositive, fatherId=fReference[0]}
  [3644] = {x=-201.504, y=147.9, z=44, rx=180, rz=-147.619, shoulder=lefty, elbow=epositive, wrist=wpositive, fatherId=fReference[0]}
  [3645] = {x=-200.213, y=147.082, z=44, rx=180, rz=-147.542, shoulder=lefty, elbow=epositive, wrist=wpositive, fatherId=fReference[0]}
  [3646] = {x=-198.923, y=146.261, z=44, rx=180, rz=-147.467, shoulder=lefty, elbow=epositive, wrist=wpositive, fatherId=fReference[0]}
  [3647] = {x=-197.633, y=145.438, z=44, rx=-180, rz=-147.391, shoulder=lefty, elbow=epositive, wrist=wpositive, fatherId=fReference[0]}
  [3648] = {x=-196.344, y=144.614, z=44, rx=-180, rz=-147.317, shoulder=lefty, elbow=epositive, wrist=wpositive, fatherId=fReference[0]}
  [3649] = {x=-195.055, y=143.787, z=44, rx=-180, rz=-147.242, shoulder=lefty, elbow=epositive, wrist=wpositive, fatherId=fReference[0]}
  [3650] = {x=-193.768, y=142.958, z=44, rx=-180, rz=-147.169, shoulder=lefty, elbow=epositive, wrist=wpositive, fatherId=fReference[0]}
  [3651] = {x=-192.48, y=142.128, z=44, rx=-180, rz=-147.096, shoulder=lefty, elbow=epositive, wrist=wpositive, fatherId=fReference[0]}
  [3652] = {x=-191.194, y=141.295, z=44, rx=-180, rz=-147.024, shoulder=lefty, elbow=epositive, wrist=wpositive, fatherId=fReference[0]}
  [3653] = {x=-189.908, y=140.461, z=44, rx=-180, rz=-146.952, shoulder=lefty, elbow=epositive, wrist=wpositive, fatherId=fReference[0]}
  [3654] = {x=-188.622, y=139.625, z=44, rx=180, rz=-146.88, shoulder=lefty, elbow=epositive, wrist=wpositive, fatherId=fReference[0]}
  [3655] = {x=-187.337, y=138.786, z=44, rx=180, rz=-146.81, shoulder=lefty, elbow=epositive, wrist=wpositive, fatherId=fReference[0]}
  [3656] = {x=-186.053, y=137.946, z=44, rx=180, rz=-146.74, shoulder=lefty, elbow=epositive, wrist=wpositive, fatherId=fReference[0]}
  [3657] = {x=-184.769, y=137.104, z=44, rx=180, rz=-146.67, shoulder=lefty, elbow=epositive, wrist=wpositive, fatherId=fReference[0]}
  [3658] = {x=-183.486, y=136.26, z=44, rx=180, rz=-146.601, shoulder=lefty, elbow=epositive, wrist=wpositive, fatherId=fReference[0]}
  [3659] = {x=-182.204, y=135.415, z=44, rx=-180, rz=-146.533, shoulder=lefty, elbow=epositive, wrist=wpositive, fatherId=fReference[0]}
  [3660] = {x=-180.922, y=134.567, z=44, rx=180, rz=-146.465, shoulder=lefty, elbow=epositive, wrist=wpositive, fatherId=fReference[0]}
  [3661] = {x=-179.641, y=133.718, z=44, rx=-180, rz=-146.398, shoulder=lefty, elbow=epositive, wrist=wpositive, fatherId=fReference[0]}
  [3662] = {x=-178.36, y=132.867, z=44, rx=-180, rz=-146.331, shoulder=lefty, elbow=epositive, wrist=wpositive, fatherId=fReference[0]}
  [3663] = {x=-177.08, y=132.014, z=44, rx=-180, rz=-146.265, shoulder=lefty, elbow=epositive, wrist=wpositive, fatherId=fReference[0]}
  [3664] = {x=-175.8, y=131.16, z=44, rx=180, rz=-146.199, shoulder=lefty, elbow=epositive, wrist=wpositive, fatherId=fReference[0]}
  [3665] = {x=-174.521, y=130.304, z=44, rx=-180, rz=-146.134, shoulder=lefty, elbow=epositive, wrist=wpositive, fatherId=fReference[0]}
  [3666] = {x=-173.242, y=129.446, z=44, rx=-180, rz=-146.07, shoulder=lefty, elbow=epositive, wrist=wpositive, fatherId=fReference[0]}
  [3667] = {x=-171.964, y=128.586, z=44, rx=180, rz=-146.006, shoulder=lefty, elbow=epositive, wrist=wpositive, fatherId=fReference[0]}
  [3668] = {x=-170.687, y=127.724, z=44, rx=-180, rz=-145.943, shoulder=lefty, elbow=epositive, wrist=wpositive, fatherId=fReference[0]}
  [3669] = {x=-169.41, y=126.861, z=44, rx=-180, rz=-145.88, shoulder=lefty, elbow=epositive, wrist=wpositive, fatherId=fReference[0]}
  [3670] = {x=-168.134, y=125.996, z=44, rx=180, rz=-145.818, shoulder=lefty, elbow=epositive, wrist=wpositive, fatherId=fReference[0]}
  [3671] = {x=-166.858, y=125.13, z=44, rx=-180, rz=-145.756, shoulder=lefty, elbow=epositive, wrist=wpositive, fatherId=fReference[0]}
  [3672] = {x=-165.583, y=124.262, z=44, rx=-180, rz=-145.695, shoulder=lefty, elbow=epositive, wrist=wpositive, fatherId=fReference[0]}
  [3673] = {x=-164.308, y=123.392, z=44, rx=180, rz=-145.634, shoulder=lefty, elbow=epositive, wrist=wpositive, fatherId=fReference[0]}
  [3674] = {x=-163.034, y=122.521, z=44, rx=-180, rz=-145.574, shoulder=lefty, elbow=epositive, wrist=wpositive, fatherId=fReference[0]}
  [3675] = {x=-161.76, y=121.648, z=44, rx=180, rz=-145.515, shoulder=lefty, elbow=epositive, wrist=wpositive, fatherId=fReference[0]}
  [3676] = {x=-160.487, y=120.773, z=44, rx=-180, rz=-145.455, shoulder=lefty, elbow=epositive, wrist=wpositive, fatherId=fReference[0]}
  [3677] = {x=-159.215, y=119.897, z=44, rx=-180, rz=-145.397, shoulder=lefty, elbow=epositive, wrist=wpositive, fatherId=fReference[0]}
  [3678] = {x=-157.942, y=119.02, z=44, rx=180, rz=-145.339, shoulder=lefty, elbow=epositive, wrist=wpositive, fatherId=fReference[0]}
  [3679] = {x=-156.671, y=118.141, z=44, rx=-180, rz=-145.282, shoulder=lefty, elbow=epositive, wrist=wpositive, fatherId=fReference[0]}
  [3680] = {x=-155.4, y=117.26, z=44, rx=-180, rz=-145.225, shoulder=lefty, elbow=epositive, wrist=wpositive, fatherId=fReference[0]}
  [3681] = {x=-154.129, y=116.378, z=44, rx=180, rz=-145.168, shoulder=lefty, elbow=epositive, wrist=wpositive, fatherId=fReference[0]}
  [3682] = {x=-152.859, y=115.494, z=44, rx=180, rz=-145.113, shoulder=lefty, elbow=epositive, wrist=wpositive, fatherId=fReference[0]}
  [3683] = {x=-151.59, y=114.609, z=44, rx=-180, rz=-145.057, shoulder=lefty, elbow=epositive, wrist=wpositive, fatherId=fReference[0]}
  [3684] = {x=-150.321, y=113.722, z=44, rx=-180, rz=-145.002, shoulder=lefty, elbow=epositive, wrist=wpositive, fatherId=fReference[0]}
  [3685] = {x=-149.052, y=112.834, z=44, rx=-180, rz=-144.948, shoulder=lefty, elbow=epositive, wrist=wpositive, fatherId=fReference[0]}
  [3686] = {x=-147.784, y=111.944, z=44, rx=-180, rz=-144.894, shoulder=lefty, elbow=epositive, wrist=wpositive, fatherId=fReference[0]}
  [3687] = {x=-146.517, y=111.053, z=44, rx=180, rz=-144.841, shoulder=lefty, elbow=epositive, wrist=wpositive, fatherId=fReference[0]}
  [3688] = {x=-145.25, y=110.161, z=44, rx=180, rz=-144.789, shoulder=lefty, elbow=epositive, wrist=wpositive, fatherId=fReference[0]}
  [3689] = {x=-143.983, y=109.267, z=44, rx=-180, rz=-144.736, shoulder=lefty, elbow=epositive, wrist=wpositive, fatherId=fReference[0]}
  [3690] = {x=-142.717, y=108.372, z=44, rx=-180, rz=-144.685, shoulder=lefty, elbow=epositive, wrist=wpositive, fatherId=fReference[0]}
  [3691] = {x=-141.452, y=107.475, z=44, rx=-180, rz=-144.634, shoulder=lefty, elbow=epositive, wrist=wpositive, fatherId=fReference[0]}
  [3692] = {x=-140.187, y=106.578, z=44, rx=-180, rz=-144.583, shoulder=lefty, elbow=epositive, wrist=wpositive, fatherId=fReference[0]}
  [3693] = {x=-138.922, y=105.678, z=44, rx=-180, rz=-144.533, shoulder=lefty, elbow=epositive, wrist=wpositive, fatherId=fReference[0]}
  [3694] = {x=-137.658, y=104.778, z=44, rx=-180, rz=-144.483, shoulder=lefty, elbow=epositive, wrist=wpositive, fatherId=fReference[0]}
  [3695] = {x=-136.395, y=103.876, z=44, rx=-180, rz=-144.434, shoulder=lefty, elbow=epositive, wrist=wpositive, fatherId=fReference[0]}
  [3696] = {x=-135.131, y=102.973, z=44, rx=180, rz=-144.385, shoulder=lefty, elbow=epositive, wrist=wpositive, fatherId=fReference[0]}
  [3697] = {x=-133.869, y=102.068, z=44, rx=180, rz=-144.337, shoulder=lefty, elbow=epositive, wrist=wpositive, fatherId=fReference[0]}
  [3698] = {x=-132.606, y=101.162, z=44, rx=-180, rz=-144.29, shoulder=lefty, elbow=epositive, wrist=wpositive, fatherId=fReference[0]}
  [3699] = {x=-131.345, y=100.255, z=44, rx=180, rz=-144.242, shoulder=lefty, elbow=epositive, wrist=wpositive, fatherId=fReference[0]}
  [3700] = {x=-130.083, y=99.347, z=44, rx=180, rz=-144.196, shoulder=lefty, elbow=epositive, wrist=wpositive, fatherId=fReference[0]}
  [3701] = {x=-128.822, y=98.437, z=44, rx=-180, rz=-144.15, shoulder=lefty, elbow=epositive, wrist=wpositive, fatherId=fReference[0]}
  [3702] = {x=-127.562, y=97.527, z=44, rx=180, rz=-144.104, shoulder=lefty, elbow=epositive, wrist=wpositive, fatherId=fReference[0]}
  [3703] = {x=-126.302, y=96.615, z=44, rx=-180, rz=-144.059, shoulder=lefty, elbow=epositive, wrist=wpositive, fatherId=fReference[0]}
  [3704] = {x=-125.042, y=95.702, z=44, rx=-180, rz=-144.014, shoulder=lefty, elbow=epositive, wrist=wpositive, fatherId=fReference[0]}
  [3705] = {x=-123.783, y=94.787, z=44, rx=180, rz=-143.97, shoulder=lefty, elbow=epositive, wrist=wpositive, fatherId=fReference[0]}
  [3706] = {x=-122.525, y=93.872, z=44, rx=180, rz=-143.926, shoulder=lefty, elbow=epositive, wrist=wpositive, fatherId=fReference[0]}
  [3707] = {x=-121.266, y=92.955, z=44, rx=180, rz=-143.883, shoulder=lefty, elbow=epositive, wrist=wpositive, fatherId=fReference[0]}
  [3708] = {x=-120.009, y=92.037, z=44, rx=-180, rz=-143.841, shoulder=lefty, elbow=epositive, wrist=wpositive, fatherId=fReference[0]}
  [3709] = {x=-118.751, y=91.118, z=44, rx=-180, rz=-143.798, shoulder=lefty, elbow=epositive, wrist=wpositive, fatherId=fReference[0]}
  [3710] = {x=-117.494, y=90.198, z=44, rx=180, rz=-143.757, shoulder=lefty, elbow=epositive, wrist=wpositive, fatherId=fReference[0]}
  [3711] = {x=-116.238, y=89.277, z=44, rx=180, rz=-143.715, shoulder=lefty, elbow=epositive, wrist=wpositive, fatherId=fReference[0]}
  [3712] = {x=-114.981, y=88.355, z=44, rx=180, rz=-143.675, shoulder=lefty, elbow=epositive, wrist=wpositive, fatherId=fReference[0]}
  [3713] = {x=-113.726, y=87.432, z=44, rx=-180, rz=-143.634, shoulder=lefty, elbow=epositive, wrist=wpositive, fatherId=fReference[0]}
  [3714] = {x=-112.47, y=86.507, z=44, rx=-180, rz=-143.595, shoulder=lefty, elbow=epositive, wrist=wpositive, fatherId=fReference[0]}
  [3715] = {x=-111.215, y=85.582, z=44, rx=180, rz=-143.555, shoulder=lefty, elbow=epositive, wrist=wpositive, fatherId=fReference[0]}
  [3716] = {x=-109.961, y=84.656, z=44, rx=180, rz=-143.516, shoulder=lefty, elbow=epositive, wrist=wpositive, fatherId=fReference[0]}
  [3717] = {x=-108.707, y=83.728, z=44, rx=180, rz=-143.478, shoulder=lefty, elbow=epositive, wrist=wpositive, fatherId=fReference[0]}
  [3718] = {x=-107.453, y=82.8, z=44, rx=-180, rz=-143.44, shoulder=lefty, elbow=epositive, wrist=wpositive, fatherId=fReference[0]}
  [3719] = {x=-106.2, y=81.87, z=44, rx=-180, rz=-143.403, shoulder=lefty, elbow=epositive, wrist=wpositive, fatherId=fReference[0]}
  [3720] = {x=-104.947, y=80.94, z=44, rx=180, rz=-143.366, shoulder=lefty, elbow=epositive, wrist=wpositive, fatherId=fReference[0]}
  [3721] = {x=-103.694, y=80.008, z=44, rx=-180, rz=-143.329, shoulder=lefty, elbow=epositive, wrist=wpositive, fatherId=fReference[0]}
  [3722] = {x=-102.442, y=79.076, z=44, rx=-180, rz=-143.293, shoulder=lefty, elbow=epositive, wrist=wpositive, fatherId=fReference[0]}
  [3723] = {x=-101.19, y=78.143, z=44, rx=180, rz=-143.258, shoulder=lefty, elbow=epositive, wrist=wpositive, fatherId=fReference[0]}
  [3724] = {x=-99.938, y=77.208, z=44, rx=-180, rz=-143.223, shoulder=lefty, elbow=epositive, wrist=wpositive, fatherId=fReference[0]}
  [3725] = {x=-98.687, y=76.273, z=44, rx=-180, rz=-143.188, shoulder=lefty, elbow=epositive, wrist=wpositive, fatherId=fReference[0]}
  [3726] = {x=-97.437, y=75.337, z=44, rx=-180, rz=-143.154, shoulder=lefty, elbow=epositive, wrist=wpositive, fatherId=fReference[0]}
  [3727] = {x=-96.186, y=74.4, z=44, rx=-180, rz=-143.12, shoulder=lefty, elbow=epositive, wrist=wpositive, fatherId=fReference[0]}
  [3728] = {x=-94.936, y=73.462, z=44, rx=-180, rz=-143.087, shoulder=lefty, elbow=epositive, wrist=wpositive, fatherId=fReference[0]}
  [3729] = {x=-93.686, y=72.523, z=44, rx=-180, rz=-143.054, shoulder=lefty, elbow=epositive, wrist=wpositive, fatherId=fReference[0]}
  [3730] = {x=-92.437, y=71.584, z=44, rx=-180, rz=-143.022, shoulder=lefty, elbow=epositive, wrist=wpositive, fatherId=fReference[0]}
  [3731] = {x=-91.188, y=70.643, z=44, rx=180, rz=-142.99, shoulder=lefty, elbow=epositive, wrist=wpositive, fatherId=fReference[0]}
  [3732] = {x=-89.939, y=69.702, z=44, rx=-180, rz=-142.959, shoulder=lefty, elbow=epositive, wrist=wpositive, fatherId=fReference[0]}
  [3733] = {x=-88.691, y=68.76, z=44, rx=-180, rz=-142.928, shoulder=lefty, elbow=epositive, wrist=wpositive, fatherId=fReference[0]}
  [3734] = {x=-87.443, y=67.817, z=44, rx=-180, rz=-142.897, shoulder=lefty, elbow=epositive, wrist=wpositive, fatherId=fReference[0]}
  [3735] = {x=-86.195, y=66.873, z=44, rx=180, rz=-142.867, shoulder=lefty, elbow=epositive, wrist=wpositive, fatherId=fReference[0]}
  [3736] = {x=-84.948, y=65.929, z=44, rx=-180, rz=-142.838, shoulder=lefty, elbow=epositive, wrist=wpositive, fatherId=fReference[0]}
  [3737] = {x=-83.701, y=64.984, z=44, rx=-180, rz=-142.809, shoulder=lefty, elbow=epositive, wrist=wpositive, fatherId=fReference[0]}
  [3738] = {x=-82.454, y=64.038, z=44, rx=180, rz=-142.78, shoulder=lefty, elbow=epositive, wrist=wpositive, fatherId=fReference[0]}
  [3739] = {x=-81.208, y=63.091, z=44, rx=-180, rz=-142.752, shoulder=lefty, elbow=epositive, wrist=wpositive, fatherId=fReference[0]}
  [3740] = {x=-79.962, y=62.143, z=44, rx=-180, rz=-142.724, shoulder=lefty, elbow=epositive, wrist=wpositive, fatherId=fReference[0]}
  [3741] = {x=-78.716, y=61.195, z=44, rx=-180, rz=-142.697, shoulder=lefty, elbow=epositive, wrist=wpositive, fatherId=fReference[0]}
  [3742] = {x=-77.47, y=60.246, z=44, rx=-180, rz=-142.67, shoulder=lefty, elbow=epositive, wrist=wpositive, fatherId=fReference[0]}
  [3743] = {x=-76.225, y=59.297, z=44, rx=-180, rz=-142.644, shoulder=lefty, elbow=epositive, wrist=wpositive, fatherId=fReference[0]}
  [3744] = {x=-74.98, y=58.346, z=44, rx=-180, rz=-142.618, shoulder=lefty, elbow=epositive, wrist=wpositive, fatherId=fReference[0]}
  [3745] = {x=-73.736, y=57.395, z=44, rx=-180, rz=-142.592, shoulder=lefty, elbow=epositive, wrist=wpositive, fatherId=fReference[0]}
  [3746] = {x=-72.491, y=56.444, z=44, rx=-180, rz=-142.567, shoulder=lefty, elbow=epositive, wrist=wpositive, fatherId=fReference[0]}
  [3747] = {x=-71.247, y=55.491, z=44, rx=-180, rz=-142.543, shoulder=lefty, elbow=epositive, wrist=wpositive, fatherId=fReference[0]}
  [3748] = {x=-70.003, y=54.538, z=44, rx=180, rz=-142.518, shoulder=lefty, elbow=epositive, wrist=wpositive, fatherId=fReference[0]}
  [3749] = {x=-68.76, y=53.585, z=44, rx=-180, rz=-142.495, shoulder=lefty, elbow=epositive, wrist=wpositive, fatherId=fReference[0]}
  [3750] = {x=-67.516, y=52.63, z=44, rx=-180, rz=-142.471, shoulder=lefty, elbow=epositive, wrist=wpositive, fatherId=fReference[0]}
  [3751] = {x=-66.273, y=51.676, z=44, rx=-180, rz=-142.449, shoulder=lefty, elbow=epositive, wrist=wpositive, fatherId=fReference[0]}
  [3752] = {x=-65.03, y=50.72, z=44, rx=180, rz=-142.426, shoulder=lefty, elbow=epositive, wrist=wpositive, fatherId=fReference[0]}
  [3753] = {x=-63.788, y=49.764, z=44, rx=-180, rz=-142.404, shoulder=lefty, elbow=epositive, wrist=wpositive, fatherId=fReference[0]}
  [3754] = {x=-62.545, y=48.808, z=44, rx=180, rz=-142.383, shoulder=lefty, elbow=epositive, wrist=wpositive, fatherId=fReference[0]}
  [3755] = {x=-61.303, y=47.85, z=44, rx=-180, rz=-142.362, shoulder=lefty, elbow=epositive, wrist=wpositive, fatherId=fReference[0]}
  [3756] = {x=-60.061, y=46.893, z=44, rx=-180, rz=-142.341, shoulder=lefty, elbow=epositive, wrist=wpositive, fatherId=fReference[0]}
  [3757] = {x=-58.82, y=45.934, z=44, rx=-180, rz=-142.321, shoulder=lefty, elbow=epositive, wrist=wpositive, fatherId=fReference[0]}
